	//--------------------------
	//2te Spur am Tag
	//--------------------------
	  //Begin ---------------------------------------------------------------------------------------
	    IF "DB_Schaltuhr".Tag_aktiv[#i].AZ_Begin2_aktiv = true THEN //Wenn Zeit aktiv
	    
	        #Array[#j].Min := TOD_TO_DINT(DTL_TO_TOD("DB_Schaltuhr".Tag[#i].AZ_Begin2))/60000+(#i-1)*1440; //Kopiere im Array
	    #j := #j + 1; //Array+1
	    #pruef := #pruef + 1;
	    
	    IF #anfang = 0 THEN
	        #anfang := 1;
	    END_IF;
	    
	    IF #pruef <> 1 THEN
	        #Error := true;
	    END_IF;
	    
	    END_IF;
	    //Ende ------------------------------------------------------------------------------------------
	    
	    //Begin ---------------------------------------------------------------------------------------
	    IF "DB_Schaltuhr".Tag_aktiv[#i].AZ_Ende2_aktiv = true THEN//Wenn Zeit aktiv
	    
	        #Array[#j].Min := TOD_TO_DINT(DTL_TO_TOD("DB_Schaltuhr".Tag[#i].AZ_Ende2))/60000+(#i-1)* 1440;//Kopiere im Array
	    #j := #j + 1;//Array+1
	    #pruef := #pruef - 1;
	    
	    IF #anfang = 0 THEN
	        #anfang := -1;
	        #pruef := 0; //Pruefparameter wieder auf Null
	    END_IF;
	    
	    IF #pruef <> 0 THEN
	        #Error := true;
	    END_IF;
	    
	    END_IF;
	    //Ende ------------------------------------------------------------------------------------------
	
	 END_FOR;
	 
	//Array schließen ----------------------------
	#Array[#j].Min := -1; //Ende des Arrays
	
	//Plausibilitätsprüfung
	FOR #i:=0 TO #j-2 DO
	  IF #Array[#i+1].Min<=#Array[#i].Min THEN
	    #Error:=true;
	    END_IF;
	  END_FOR;
	
	  IF #anfang = 1 AND #pruef <> 0 OR #anfang = -1 AND #pruef <> 1 OR #anfang=0 THEN //Letzte prüfung
	      #Error := true;
	    END_IF;
	    
	  IF #anfang = -1 THEN //Start mit Ausschaltung
	      #Start_Aus := true;
	  END_IF;
	
	END_IF;
	
END_FUNCTION

FUNCTION_BLOCK "Uhrzeit_WSU"
{ S7_Optimized_Access := 'FALSE' }
VERSION : 0.1
   VAR 
      aktDatum {InstructionName := 'DTL'; LibVersion := '1.0'} : DTL;
      Time_to_on : Int;   // Zeit bis/seit Arbeitszeitbeginn Wert>0-->bis Wert<0-->seit (in Minuten]
      Time_to_off : Int;   // Zeit bis/seit Arbeitszeitende Wert>0-->bis Wert<0-->seit (in Minuten]
      min_of_week : Int;   // Minuten seit Wochenbeginn
      BA_Uhr_Ein : Bool;   // Dauer-Ein BA_Uhr_Aus: 9.0=0 UND 9.1=0
      BA_Uhr_Dauer : Bool;   // Uhrenbetrieb
      AZ_aktiv : Bool;   // Arbeitszeit aktiv
      ProfileWeek : Array[0..28] of Struct   // Wochenschaltpunkte
         MinWeek : Int;
         State : Byte;   // 0=kein Eintrag, bit0=ein, bit1=aus
         resB : Byte;
      END_STRUCT;
   END_VAR

   VAR_TEMP 
      retVal : Int;
      Woko : DInt;   // muss direkt hinter ProfileWeek stehen!
      rdRetval : Int;
      WoTime_bis : Int;
      WoTime_seit : Int;
      TempTime : Int;
      lastOn : Bool;
      nextOn : Bool;
      lastFnd : Bool;
      nextFnd : Bool;
      i : Int;
   END_VAR

   VAR CONSTANT 
      MaxWeek : Int := 10080;   // Anzahl Minuten pro Woche
      "0x7FFF" : Int := 32767;
   END_VAR


BEGIN
	//Lokalzeit auslesen
	IF RD_LOC_T(#aktDatum) > #"0x7FFF"  THEN //Wenn Retval >= 0x08000,
	    RETURN;
	END_IF;
	
	//-------------
	//Betriebsart
	//-------------
	
	//-----------------------------
	//Uhrenbetrieb (Wochenfunktion)
	//-----------------------------
	IF #BA_Uhr_Ein THEN
	    REGION Woche
	        #lastFnd := FALSE;  //letzter Eintrag gefunden/Wochenwechsel erkannt
	        #nextFnd := FALSE;  //nächster Eintrag gefunden
	        #lastOn := FALSE;
	        #nextOn := FALSE;
	        
	        #WoTime_bis := 32767;
	        #WoTime_seit := 32767;
	        
	        //--------------------------------------------------------------------------
	        //Berechnung Minuten seit Wochenbeginn
	        //--------------------------------------------------------------------------
	        #min_of_week := ((USINT_TO_INT(#aktDatum.WEEKDAY) - 1) * 1440) + (USINT_TO_INT(#aktDatum.HOUR) * 60) + USINT_TO_INT(#aktDatum.MINUTE); //Wenn aktueller Wochentag 1 = Sonntag
	        
	        //Schaltuhr leer?
	        IF #ProfileWeek[1].State = b#16#0 THEN
	            #Time_to_on := 32767;
	            #Time_to_off := -32767;
	            
	            //----------------------------
	            //Schaltpunkte suchen
	            //----------------------------
	        ELSE
	            
	            //--------------------------------------------------------------------------
	            //letzten Schaltpunkt suchen
	            //--------------------------------------------------------------------------
	        REGION last
	            //alles ab rela:
	            //vorherigen Schaltpunkt suchen
	                #Woko := #min_of_week;
	                #i := -1;
	                
	                REPEAT //FOR Schleife geht nicht weil ich #i während des Ablaufs nicht verändern darf :-(
	                    
	                    #i += 1;
	                    
	                    IF #ProfileWeek[#i].State <> 0 AND #Woko >= #ProfileWeek[#i].MinWeek THEN //Eintrag leer oder in der Zukunft? dann weiter
	                        //Eintrag gefunden
	                        #lastFnd := TRUE;
	                        IF #ProfileWeek[#i].State = 1 THEN
	                            #lastOn := TRUE;
	                        ELSIF #ProfileWeek[#i].State = 2 THEN
	                            #lastOn := FALSE;
	                        END_IF;
	                        
	                        IF #min_of_week < #ProfileWeek[#i].MinWeek THEN
	                            #WoTime_seit := #MaxWeek - #ProfileWeek[#i].MinWeek + #min_of_week;
	                        ELSE
	                            #WoTime_seit := #min_of_week - #ProfileWeek[#i].MinWeek;
	                        END_IF;
	                    END_IF;
	                    
	                //Prüfung im letzten Durchgang
	                IF #i = 28 THEN
	                    //fündig geworden?
	                    IF #lastFnd THEN//gefunden, ok
	                        EXIT;
	                        
	                    //keinen letzten Schaltpunkt entdeckt
	                    //aktueller Status bleibt erhalten
	                    ELSIF #Woko = #MaxWeek THEN //im 2ten Durchgang?
	                        IF #Time_to_on < 0 THEN
	                            #lastOn := TRUE;
	                            #WoTime_seit := #Time_to_on * -1;
	                        ELSE
	                            #lastOn := FALSE;
	                            #WoTime_seit := #Time_to_off * -1;
	                        END_IF;
	                        
	                        EXIT;
	                        
	                    ELSE//im ersten Durchgang nichts gefunden, dann evtl. in voriger Woche im 2ten Durchgang?
	                        #Woko := #MaxWeek;
	                        #i := -1;
	                    END_IF;
	                END_IF;
	                
	            UNTIL #i = 28
	            END_REPEAT;
	        END_REGION
	            
	            //--------------------------------------------------------------------------
	            //nächsten Schaltpunkt suchen
	            //--------------------------------------------------------------------------
	        REGION next
	            //alles ab snex:
	            //nächsten Schaltpunkt suchen
	            #i := -1;
	            
	            REPEAT //FOR Schleife geht nicht weil ich #i während des Ablaufs nicht verändern darf :-(
	                
	                #i += 1;
	                
	                IF #ProfileWeek[#i].State <> 0 AND #ProfileWeek[#i].MinWeek - #min_of_week >= 0 THEN //Eintrag leer oder in der Zukunft? dann weiter
	                    //Eintrag gefunden
	                    #TempTime := #ProfileWeek[#i].MinWeek - #min_of_week;
	                    
	                    #nextFnd := TRUE;
	                    
	                    IF #TempTime > #WoTime_bis THEN
	                        EXIT;
	                    END_IF;
	                    
	                    #WoTime_bis := #TempTime;
	                    
	                    IF #ProfileWeek[#i].State = 1 THEN
	                        #nextOn := TRUE;
	                    ELSIF #ProfileWeek[#i].State = 2 THEN
	                        #nextOn := FALSE;
	                    END_IF;
	                    EXIT;
	                    
	                END_IF;
	                
	            UNTIL #i = 28
	            END_REPEAT;
	            
	            //nichts gefunden? Dann nächste Woche checken (ersten Eintrag)
	            //Prüfung im letzten Durchgang
	            IF NOT #nextFnd THEN
	                #TempTime := #MaxWeek - #min_of_week + #ProfileWeek[0].MinWeek;
	                #nextFnd := TRUE;
	                IF #TempTime <= #WoTime_bis THEN
	                    #WoTime_bis := #TempTime;
	                    
	                    IF #ProfileWeek[0].State = 1 THEN
	                        #nextOn := TRUE;
	                    ELSIF #ProfileWeek[0].State = 2 THEN
	                        #nextOn := FALSE;
	                    END_IF;
	                END_IF;
	            END_IF;
	            
	        END_REGION
	        
	            END_IF;
	            
	            //Auswertung zum Schluss
	            IF #lastOn AND #nextOn THEN
	                #Time_to_on := 0;// -32767;
	                #Time_to_off := 32767;
	            ELSIF NOT #lastOn AND NOT #nextOn THEN
	                #Time_to_on := 32767;
	                #Time_to_off := 0;// -32767;
	            ELSIF #lastOn AND NOT #nextOn THEN
	                #Time_to_off := #WoTime_bis;
	                #Time_to_on := #WoTime_seit * -1;
	            ELSE
	                #Time_to_on := #WoTime_bis;
	                #Time_to_off := #WoTime_seit * -1;
	            END_IF;
	            
	            
	            
	    END_REGION
	    
	//-----------------------------   
	//Dauerbetrieb
	//-----------------------------
	ELSIF #BA_Uhr_Dauer THEN
	    REGION Dauer
	        #Time_to_on := -32767;
	        #Time_to_off := 32767;
	    END_REGION
	    
	//-----------------------------
	//Aus
	//-----------------------------
	ELSE
	    REGION Aus
	        #Time_to_on := 32767;
	        #Time_to_off := -32767;
	    END_REGION
	END_IF;
	
	//Auswertung Arbeitszeit
	#AZ_aktiv := #Time_to_on <= 0;
	
END_FUNCTION_BLOCK

FUNCTION "Komm_PNOZ" : Void   // FC360, STL
TITLE = Kommunikation Pilz-PNOZ <--> PLC
{ S7_Optimized_Access := 'FALSE' }
// stored: AutoNumber false
   VAR_TEMP
      Checksum : Word;
      ReturnValue : Int;
      count : Byte;
   END_VAR
BEGIN

NETWORK
TITLE = Aktivierung der Kommunikation

      AN    "DB_PNOZ_Comm".connection.activate;
      A     "E_T_ErrQ";
      S     "DB_PNOZ_Comm".connection.activate;


NETWORK
TITLE = OUTPUT --> PNOZ
// siehe Handbuch
// "PNOZmulti_2_Com_Interf_Man_1002971-de-03.pdf"
// Set Header   (Kap. 5.5)
      L     16#05;
      T     "DB_PNOZ_IN_Out".Out.Header[0];

      L     16#15;
      T     "DB_PNOZ_IN_Out".Out.Header[1];

      L     16#00;
      T     "DB_PNOZ_IN_Out".Out.Header[2];

      L     16#26;  // Anzahl Nutzdaten +5  = 38 dez
      T     "DB_PNOZ_IN_Out".Out.Header[3];

      L     16#5C;  // Anforderungs-Nr
      T     "DB_PNOZ_IN_Out".Out.Header[4];

      L     16#00;
      T     "DB_PNOZ_IN_Out".Out.Header[5];  // Control Byte Bit 0..2 Watchdog

      L     16#00;
      T     "DB_PNOZ_IN_Out".Out.Header[6];

      L     16#00;  // immer 0x00
      T     "DB_PNOZ_IN_Out".Out.Header[7];

      L     16#10;
      T     "DB_PNOZ_IN_Out".Out.Endekennung;

// Set Vitual OUTput - je nach Projekt
      A     "E_T_Q_Not-Halt";
// alle Schütze müssen abgefallen sein
      A     "E_RM_NH_Dkl";
      A     "E_RM_NH_FP_CM01.GP01";
      A     "E_RM_NH_FP_CM01.GP04";
      A     "E_RM_NH_Pumpen";
      =     "DB_PNOZ_IN_Out".Out.T_NH_Quitt;
// Freigabe Automatik
      A     "E_Frg_Auto";
      =     "DB_PNOZ_IN_Out".Out.Frg_Automatik;

      CLR;
      =     "DB_PNOZ_IN_Out".Out.VirtualOutput[16];
// ...
      =     "DB_PNOZ_IN_Out".Out.VirtualOutput[127];

// Berechnung der Checksumme (4+ .. 39)

      LAR1  P#48.0;  // fix 44 (IN) + 4

      L     "DB_PNOZ_IN_Out".Out.Header[4];  //Start
      T     #Checksum;

      L     35;  // fix: 39 - 4
T_CS: T     #count;
      OPN   "DB_PNOZ_IN_Out";
      +AR1  P#1.0;
      L     #Checksum;
      L     DBB [AR1, P#0.0];
      +I;
      T     #Checksum;

      L     #count;  //Schleifenzähler
      LOOP  T_CS;

      L     16#00;
      L     #Checksum;
      AW    16#00FF;
      -I;
      T     "DB_PNOZ_IN_Out".Out.Checksum;



NETWORK
TITLE = Umkopieren
// Sende-/Empfangsdaten umkopieren

      A     "DB_PNOZ_Comm".RECEIVE.NDR;
      R     "DB_PNOZ_Comm".RECEIVE.NDR;
      JCN   Send;

      CALL  BLKMOV
      ( SRCBLK  := "DB_PNOZ_Receive".In,
        RET_VAL := #ReturnValue,
        DSTBLK  := "DB_PNOZ_IN_Out".In
      );

Send: A     "DB_PNOZ_Comm".SEND.Busy;
      JC    no_Send_DATA;

      CALL  BLKMOV
      ( SRCBLK  := "DB_PNOZ_IN_Out".Out,
        RET_VAL := #ReturnValue,
        DSTBLK  := "DB_PNOZ_Send".Out
      );

no_Send_DATA:NOP   0;

NETWORK
TITLE = Sprungverteiler

      L     "DB_PNOZ_Comm".Global_Status;
      JL    LSTX;
      JU    OFF;  // 0: Aus
      JU    CONN;  // 1: Verbindungsaufbau
      JU    WRIT;  // 2: Schreiben
      JU    READ;  // 3: Lesen
      JU    DISC;  // 4:Verbindungsabbau
      JU    ERR;  // 5: Fehler
LSTX: JU    ende;

//*
// wait for user input (activate / deactivate communication)
// - if activate change for 0 to 1
//    => status is set to 1 (connect) and all status-values are set to default
// - if activate change for 1 to 0
//    => status is set to 4 (disconnect)
//-

OFF:  A     "DB_PNOZ_Comm".connection.activate;
      AN    "DB_PNOZ_Comm".connection.established;
      JCN   OFF1;

// Aktivieren
      SET;
      S     "DB_PNOZ_Comm".connection.established;

      L     1;  // Verbindungsaufbau
      T     "DB_PNOZ_Comm".Global_Status;

// init
      SET;
      R     "DB_PNOZ_Comm".CONNECT.Request;
      R     "DB_PNOZ_Comm".CONNECT.Done;
      R     "DB_PNOZ_Comm".CONNECT.Error;

      R     "DB_PNOZ_Comm".SEND.Request;
      R     "DB_PNOZ_Comm".SEND.Done;
      R     "DB_PNOZ_Comm".SEND.Error;

      S     "DB_PNOZ_Comm".RECEIVE.EN_R;  // immer 1
      R     "DB_PNOZ_Comm".RECEIVE.NDR;
      R     "DB_PNOZ_Comm".RECEIVE.Error;

      R     "DB_PNOZ_Comm".DISCONNECT.Request;
      R     "DB_PNOZ_Comm".DISCONNECT.Done;
      R     "DB_PNOZ_Comm".DISCONNECT.Error;

      JU    ende;

// Deaktivieren
OFF1: AN    "DB_PNOZ_Comm".connection.activate;
      A     "DB_PNOZ_Comm".connection.established;
      JCN   ende;

      SET;
      R     "DB_PNOZ_Comm".connection.established;
      R     "DB_PNOZ_Comm".CONNECT.Done;
      R     "DB_PNOZ_Comm".SEND.Done;
      R     "DB_PNOZ_Comm".RECEIVE.NDR;

      L     4;  // Verbindungsabbau
      T     "DB_PNOZ_Comm".Global_Status;

      JU    ende;


NETWORK
TITLE = Verbindungsaufbau
// call FB65 (TCON) as long as status = 1 (connect)
//  - if connection_1 is established (TCON_DONE=1) change to status=2 (send)
//  - if an error occurs (TCON_ERR=1) change to status=5 (error)
CONN: L     2;
      T     "DB_PNOZ_Comm".CONNECT.ID;
      T     "DB_PNOZ_Comm".Connection_Param.local_device_id;

      CALL  TCON, "TCON_DI"
      ( REQ     := "DB_PNOZ_Comm".CONNECT.Request,
        ID      := "DB_PNOZ_Comm".CONNECT.ID,
        DONE    := "DB_PNOZ_Comm".CONNECT.Done,
        BUSY    := "DB_PNOZ_Comm".CONNECT.Busy,
        ERROR   := "DB_PNOZ_Comm".CONNECT.Error,
        STATUS  := "DB_PNOZ_Comm".CONNECT.Status,
        CONNECT := "PNOZ_Connection_DB"
      );

      SET;
      S     "DB_PNOZ_Comm".CONNECT.Request;

      A     "DB_PNOZ_Comm".CONNECT.Done;
      R     "DB_PNOZ_Comm".CONNECT.Done;
      R     "DB_PNOZ_Comm".SEND.Request;
      JC    to_S;

      L     "DB_PNOZ_Comm".CONNECT.Status;
      L     16#80A3;  //Verbindung gibt's schon
      ==I;
      A     "DB_PNOZ_Comm".CONNECT.Error;
      R     "DB_PNOZ_Comm".DISCONNECT.Request;
      JC    to_D;

      A     "DB_PNOZ_Comm".CONNECT.Error;
      JC    to_E;

      JU    ende;

to_S: L     2;  // --> Senden
      T     "DB_PNOZ_Comm".Global_Status;
      JU    ende;

to_D: L     4;  // --> Verbindungsabbau
      T     "DB_PNOZ_Comm".Global_Status;
      JU    ende;


to_E: L     5;  // --> Fehler
      T     "DB_PNOZ_Comm".Global_Status;

      JU    ende;


NETWORK
TITLE = Schreiben --> PNOZ
// call FB63 (TSEND) as long as status = 2 (send)
//  - if send is complete (TSEND_DONE=1) change to status=3 (receive)
//  - if an error occurs (TSEND_ERR=1)
//    - if TSEND_STATUS='80A1' or '80C4' stay at status=2 and try to send again
//    - if TSEND_STATUS<>'80A1' or '80C4' change to status=5 (error)
WRIT: L     43;  //fix PNOZ
      T     "DB_PNOZ_Comm".SEND.Length;

      L     "DB_PNOZ_Comm".CONNECT.ID;
      T     "DB_PNOZ_Comm".SEND.ID;

      CALL  TSEND, "TSEND_DI"
      ( REQ    := "DB_PNOZ_Comm".SEND.Request,
        ID     := "DB_PNOZ_Comm".SEND.ID,
        LEN    := "DB_PNOZ_Comm".SEND.Length,
        DONE   := "DB_PNOZ_Comm".SEND.Done,
        BUSY   := "DB_PNOZ_Comm".SEND.Busy,
        ERROR  := "DB_PNOZ_Comm".SEND.Error,
        STATUS := "DB_PNOZ_Comm".SEND.Status,
        DATA   := "DB_PNOZ_Send".Out
      );

      SET;
      S     "DB_PNOZ_Comm".SEND.Request;

      A     "DB_PNOZ_Comm".SEND.Done;
      R     "DB_PNOZ_Comm".SEND.Done;
      S     "DB_PNOZ_Comm".RECEIVE.EN_R;
      JC    toRV;

      L     16#80A1;  //Kommunikationsfehler
      L     "DB_PNOZ_Comm".SEND.Status;
      ==I;
      O(;
      L     16#80C4;  //Temporärer Kommunikationsfehler
      ==I;
      );
      A     "DB_PNOZ_Comm".SEND.Error;
      R     "DB_PNOZ_Comm".SEND.Request;  // --> nochmal versuchen
      JC    ende;

      A     "DB_PNOZ_Comm".SEND.Error;
      JC    SDER;

      JU    ende;

toRV: L     3;
      T     "DB_PNOZ_Comm".Global_Status;
      JU    ende;

SDER: L     5;
      T     "DB_PNOZ_Comm".Global_Status;
      JU    ende;


NETWORK
TITLE = Lesen <-- PNOZ
// call FB64 (TRCV) as long as status = 3 (receive)
//  - if new data is received (TSEND_NDR=1) change to status=2 (receive)
//    and increment send_values
//  - if an error occurs (TRCV_ERR=1)
//    - if TRCV_STATUS='80A1' or '80C4' change to status=2 and try to send
//    - if TRCV_STATUS<>'80A1' or '80C4' change to status=5 (error)
READ: L     43;  //fix PNOZ
      T     "DB_PNOZ_Comm".RECEIVE.Length;

      L     "DB_PNOZ_Comm".CONNECT.ID;
      T     "DB_PNOZ_Comm".RECEIVE.ID;

      CALL  TRCV, "TRCV_DI"
      ( EN_R     := "DB_PNOZ_Comm".RECEIVE.EN_R,
        ID       := "DB_PNOZ_Comm".RECEIVE.ID,
        LEN      := "DB_PNOZ_Comm".RECEIVE.Length,
        ADHOC    := "DB_PNOZ_Comm".RECEIVE.ADHOC,
        NDR      := "DB_PNOZ_Comm".RECEIVE.NDR,
        BUSY     := "DB_PNOZ_Comm".RECEIVE.Busy,
        ERROR    := "DB_PNOZ_Comm".RECEIVE.Error,
        STATUS   := "DB_PNOZ_Comm".RECEIVE.Status,
        RCVD_LEN := "DB_PNOZ_Comm".RECEIVE.Receive_Length,
        DATA     := "DB_PNOZ_Receive".In
      );

      A     "DB_PNOZ_Comm".RECEIVE.NDR;
      JC    toSD;

      L     16#80A1;  //Kommunikationsfehler
      L     "DB_PNOZ_Comm".RECEIVE.Status;
      ==I;
      O(;
      L     16#80C4;  //Temporärer Kommunikationsfehler
      ==I;
      );
      A     "DB_PNOZ_Comm".RECEIVE.Error;
      R     "DB_PNOZ_Comm".RECEIVE.Error;
      JC    toSD;

      A     "DB_PNOZ_Comm".RECEIVE.Error;
      JC    RVER;

      JU    ende;

toSD: L     2;
      T     "DB_PNOZ_Comm".Global_Status;
      SET;
      R     "DB_PNOZ_Comm".SEND.Request;
      JU    ende;

RVER: L     5;
      T     "DB_PNOZ_Comm".Global_Status;
      JU    ende;


NETWORK
TITLE = Verbindungsabbau
// call FB66 (TDISCON) as long as status = 4 (disconnect)
//  - if connection_1 is disconnected (TDISCON_DONE=1) change to status=0 (init)
//  - if an error occurs (TDISCON_ERR=1) change to status=5 (error)
DISC: L     "DB_PNOZ_Comm".CONNECT.ID;
      T     "DB_PNOZ_Comm".DISCONNECT.ID;

      CALL  TDISCON, "TDISCON_DI"
      ( REQ    := "DB_PNOZ_Comm".DISCONNECT.Request,
        ID     := "DB_PNOZ_Comm".DISCONNECT.ID,
        DONE   := "DB_PNOZ_Comm".DISCONNECT.Done,
        BUSY   := "DB_PNOZ_Comm".DISCONNECT.Busy,
        ERROR  := "DB_PNOZ_Comm".DISCONNECT.Error,
        STATUS := "DB_PNOZ_Comm".DISCONNECT.Status
      );

      SET;
      S     "DB_PNOZ_Comm".DISCONNECT.Request;

      A     "DB_PNOZ_Comm".DISCONNECT.Done;
      R     "DB_PNOZ_Comm".DISCONNECT.Done;
      R     "DB_PNOZ_Comm".connection.activate;
      R     "DB_PNOZ_Comm".connection.established;
      JC    to_O;

      A     "DB_PNOZ_Comm".DISCONNECT.Error;
      JC    toE;

      JU    ende;

to_O: L     0;  // --> OFF
      T     "DB_PNOZ_Comm".Global_Status;
      JU    ende;

toE:  L     5;  // --> Fehler
      T     "DB_PNOZ_Comm".Global_Status;
      JU    ende;


NETWORK
TITLE = Fehler
ERR:  SET;
      R     "DB_PNOZ_Comm".connection.activate;
      R     "DB_PNOZ_Comm".connection.established;

      L     0;  // --> OFF
      T     "DB_PNOZ_Comm".Global_Status;

ende: BE;

END_FUNCTION

FUNCTION "FC_DP_Error" : Void   // FC203, STL
TITLE = Profibusfehler melden
{ S7_Optimized_Access := 'FALSE' }
// stored: AutoNumber false
   VAR_TEMP
      RetVal : Int;
      Adresse : DWord;
      Count : Int;
      Wert_akt : Byte;
      Wert_alt : Byte;
      Err_Nr : USInt;
      Inf : Struct
         Inf1 : Byte;
         inf2 : Byte;
      END_STRUCT;
   END_VAR
BEGIN

NETWORK
TITLE = Störung/Ausfall
      AN    "DB_ANLAGE".config.Check_Profibus;  //keine Überwachung gefordert
      ON    "DB_ANLAGE".IN.Watch_Profibus;  //Überwachung nicht möglich
      BEC;
      R     "DB_DP_Error".Sammelwarnung;
      R     "DB_DP_Error".Sammelstoerung;

      A     "DB_ANLAGE".IN.PC_offline;  //kein PC-aktiv --> keine Überwachung
      BEC;

//Erstmalige Prüfung?
      AN    "DB_DP_Error".Init;
      AN    "DB_ANLAGE".IN.AMS_Restart;
      JC    norm;


NETWORK
TITLE = erstmalige Prüfung --> nur Fehlerstatus 2oder 3 senden
// Statuswert Bedeutung:
// 0: nicht projektiert & nicht vorhanden
// 1: vorhanden & ok
// 2: vorhanden aber nicht ok
// 3: projektiert aber nicht vorhanden
      SET;
      R     "DB_DP_Error".Init;

//aktuellen Status als Altstatus übernehmen
      CALL  FILL
      ( BVAL    := "DB_DP_Error".DP_Slave,
        RET_VAL := #RetVal,
        BLK     := "DB_DP_Error".Altwert
      );

//Altwert-Einträge mit Status 0,1 bleiben
//Einträge mit 2,3 werden auf 1 gesetzt
//dadurch wird bei fehlerhaften Einträgen ein Wechsel von 1 auf 2 oder 3 erkannt
//und somit erneut gemeldet
      L     0;
      L     "DB_DP_Error".HiAdr;
      ==I;
      BEC;
retC: T     #Count;
      L     1024;
      +D;
      SLD   3;
      T     #Adresse;
      OPN   "DB_DP_Error";
      L     DBB [#Adresse];
      L     1;  //Wert 0,1 bleibt erhalten
      <=I;
      JC    nexC;
      T     DBB [#Adresse];
nexC: L     #Count;
      LOOP  retC;  //Wert 2,3 mit 1 überschreiben

NETWORK
TITLE = Normalprüfung --> jede Statusänderung melden
norm: NOP   0;

      L     0;  //keine Profibusteilnehmer
      L     "DB_DP_Error".HiAdr;
      ==I;
      BEC;
reC:  T     #Count;
      SLD   3;
      T     #Adresse;
      OPN   "DB_DP_Error";
      L     DBB [#Adresse];
      T     #Wert_akt;  //"DB_DP_Error".DP_Slave[#Count]

      L     #Wert_akt;  //Warnung melden
      L     2;
      ==I;
      S     "DB_DP_Error".Sammelwarnung;
      L     #Wert_akt;  //Störung melden
      L     3;
      ==I;
      S     "DB_DP_Error".Sammelstoerung;

      L     #Count;
      +     1024;
      SLD   3;
      T     #Adresse;
      OPN   "DB_DP_Error";
      L     DBB [#Adresse];
      T     #Wert_alt;

//Statusauswertung und Änderung melden
      L     #Wert_akt;  //"DB_DP_Error".Altwert[#Count]
      L     #Wert_alt;
      ==I;
      JC    nxC;
      L     #Wert_alt;
      JL    list;
      JU    old0;
      JU    old1;
      JU    old2;
      JU    old3;
list: JU    nxC;

//Baugruppe war weder projektiert noch vorhanden
old0: L     #Wert_akt;
      T     #Err_Nr;
      JC    evt;

//Baugruppe war projektiert und vorhanden
old1: L     0;  //Wechsel auf 0 ist ok
      L     #Wert_akt;
      ==I;
      JC    nxC;
      T     #Err_Nr;
      JC    evt;

//Baugruppe war projektiert,vorhanden aber fehlerhaft
old2: L     0;  //Wechsel auf 0 ist ok
      L     #Wert_akt;
      ==I;
      JC    nxC;
      T     #Err_Nr;
      JC    evt;

//Baugruppe war projektiert aber nicht vorhanden
old3: L     0;  //Wechsel auf 0 ist ok
      L     #Wert_akt;
      ==I;
      JC    nxC;
      T     #Err_Nr;
      JC    evt;

evt:  NOP   0;
//Err_Nr 1:Station wiederkehr
//Err_Nr 2:Station nicht ok
//Err_Nr 3:Station Ausfall
      CALL  BLKMOV
      ( SRCBLK  := #Count,
        RET_VAL := #RetVal,
        DSTBLK  := #Inf
      );


      L     #Err_Nr;
      L     3;
      ==I;
      A     "DB_DP_Error".Hupe_enable;
      R     "DB_ANLAGE".config.M_Q_Hupe;

nxC:  L     #Count;
      LOOP  reC;

//aktuellen Status als Altstatus übernehmen
      CALL  FILL
      ( BVAL    := "DB_DP_Error".DP_Slave,
        RET_VAL := #RetVal,
        BLK     := "DB_DP_Error".Altwert
      );

END_FUNCTION

FUNCTION "FU_Read" : Void
{ S7_Optimized_Access := 'TRUE' }
VERSION : 0.1
   VAR_TEMP 
      i : Int;
      Ret_Value : Int;
   END_VAR


BEGIN
	IF "DB_ANLAGE".BA.Simulation THEN
	    RETURN;
	END_IF;
	
	// Pumpen
	#Ret_Value := DPRD_DAT(LADDR := "SEW-GW_UC01~Filterbeschickung_HQ01", RECORD => "FU_In_Out".FU[1].PE);
	#Ret_Value := DPRD_DAT(LADDR := "SEW-GW_UC01~Umwaelzung_CM01", RECORD => "FU_In_Out".FU[2].PE);
	#Ret_Value := DPRD_DAT(LADDR := "SEW-GW_UC01~Umwaelzung_CM03", RECORD => "FU_In_Out".FU[3].PE);
	#Ret_Value := DPRD_DAT(LADDR := "SEW-GW_UC01~Filterbeschickung_HQ02", RECORD => "FU_In_Out".FU[4].PE);
	#Ret_Value := DPRD_DAT(LADDR := "SEW-GW_UC01~Umwaelzung_CM02", RECORD => "FU_In_Out".FU[5].PE);
	#Ret_Value := DPRD_DAT(LADDR := "SEW-GW_UC01~Umwaelzung_CM04", RECORD => "FU_In_Out".FU[6].PE);
	//Ventilator
	#Ret_Value := DPRD_DAT(LADDR := "SEW-GW_UC01~Ventilator_Sperrluft", RECORD => "FU_In_Out".FU[7].PE);
	
	// QF
	#Ret_Value := DPRD_DAT(LADDR := "SEW-GW_UC06~QF_WR02", RECORD => "FU_In_Out".FU[8].PE);
	#Ret_Value := DPRD_DAT(LADDR := "SEW-GW_UC06~QF_WR03", RECORD => "FU_In_Out".FU[9].PE);
	// TW
	#Ret_Value := DPRD_DAT(LADDR := "SEW-GW_UC07~TW_Fahrt", RECORD => "FU_In_Out".FU[10].PE);
	#Ret_Value := DPRD_DAT(LADDR := "SEW-GW_UC07~TW_Hub_li_WR04", RECORD => "FU_In_Out".FU[11].PE);
	#Ret_Value := DPRD_DAT(LADDR := "SEW-GW_UC07~TW_Hub_re_WR05", RECORD => "FU_In_Out".FU[12].PE);
	
	FOR #i := 1 TO "FU_In_Out".Anzahl DO
	    IF "DB_ANLAGE".IN.Quitt_Err THEN
	        "FU_In_Out".FU[#i].Fehler := FALSE;
	    END_IF;
	    
	    "FU_In_Out".FU[#i].Fehler := "FU_In_Out".FU[#i].PE.Statusbyte.Stoer;
	    "FU_In_Out".FU[#i].AM_Fehlernummer := "FU_In_Out".FU[#i].PE.Statusbyte.Fehlernummer;
	END_FOR;
	
	
END_FUNCTION

FUNCTION "FC_INPUT" : Void   // FC210, STL
TITLE = Einlesen der physikalischen Eingänge
{ S7_Optimized_Access := 'FALSE' }
AUTHOR : RE
// stored: AutoNumber false
   VAR_TEMP
      WT_DB : Int;
      RetVal : Int;
   END_VAR
   VAR CONSTANT
      Aufgabe_KS : USInt := 1;
      Aufgabe_LS : USInt := 2;
      Aufgabe_GO : USInt := 3;
   END_VAR
BEGIN

NETWORK
TITLE = Simulation
// Adressen für Diagnose sind in der Hardware-Konfiguration
// hinterlegt und sind noch anzupassen !!!

//---------------------------------------------------
//Fehlerquittung
      A     "E_T_ErrQ";
      O     "MobilePanel".Drucktaster_K2_Push;
      FP    "DB_ANLAGE".config.FP_In_Quitt;
      =     "DB_ANLAGE".IN.Quitt_Err;
      L     s5t#500ms;
      Extend "T_ErrQuitt";

//---------------------------------------------------


NETWORK
TITLE = Einlesen Digitale Eingäne (allgemein)
ok:   SET;

      AN    "DB_PNOZ_IN_Out".In.PNOZ_OK;
      =     "DB_ANLAGE".IN.S_Not_Aus;

NoQt: SET;
      =     "DB_ANLAGE".IN.S_St_Spng;
      A     "E_T_HupeQ";
      =     "DB_ANLAGE".IN.Quitt_Hupe;
      =     "DB_Alarme".IN_Quitt_Hupe;

//Reperaturbetrieb über Schlüssel-Panel
      A     "MobilePanel".Koordinierung.%X2;
      L     S5T#2s;
      SD    "T_MobielPanel_Lebensbit_ein";

      AN    "MobilePanel".Koordinierung.%X2;
      L     S5T#2s;
      SD    "T_MobielPanel_Lebensbit_aus";

      A     "MobilePanel".Schluessel;
      S     "DB_ANLAGE".IN.Reparatur;

      AN    "MobilePanel".Schluessel;
      O     "T_MobielPanel_Lebensbit_ein";
      O     "T_MobielPanel_Lebensbit_aus";
      R     "DB_ANLAGE".IN.Reparatur;

      CLR;
      =     "DB_ANLAGE".IN.Reset;
      =     "DB_ANLAGE".IN.Lamp_Test;

      A     "E_Frg_Auto";
      O     "DB_ANLAGE".BA.Simulation;
      R     "DB_ANLAGE".IN.BA_Tipp;
      R     "DB_ANLAGE".IN.BA_Hand;
      S     "DB_ANLAGE".IN.BA_Auto;

      AN    "E_Frg_Auto";
      A     "Panel".Betriebsart.Hand;
      R     "DB_ANLAGE".IN.BA_Tipp;
      S     "DB_ANLAGE".IN.BA_Hand;
      R     "DB_ANLAGE".IN.BA_Auto;

      AN    "E_Frg_Auto";
      A     "Panel".Betriebsart.Tipp;
      S     "DB_ANLAGE".IN.BA_Tipp;
      R     "DB_ANLAGE".IN.BA_Hand;
      R     "DB_ANLAGE".IN.BA_Auto;

      A     "DB_ANLAGE".IN.BA_Auto;
      A     "Panel".Betriebsart.Automatik;
      R     "DB_ANLAGE".IN.Automat_aus;
      S     "DB_ANLAGE".IN.Automat_ein;

      AN    "E_Frg_Auto";
      ON    "Panel".Betriebsart.Automatik;
      S     "DB_ANLAGE".IN.Automat_aus;
      R     "DB_ANLAGE".IN.Automat_ein;

      L     1;
      A     "DB_ANLAGE".config.NormalB;
      =     "Panel".Betriebsmodus.Normal;
      R     "Panel".Betriebsmodus.Kombi;
      JC    A_BM;
      L     2;
      AN    "DB_ANLAGE".config.NormalB;
      =     "Panel".Betriebsmodus.Kombi;
      R     "Panel".Betriebsmodus.Normal;

A_BM: T     "Panel".Betriebsmodus.Anzeige;
// Wechsel nur bei komplett leerer Anlage
      L     "DI_FW_1".ZST.WT_DB_NR_li;
      L     0;
      ==I;
      A(;
      L     "DI_FW_1".ZST.WT_DB_NR_re;
      ==I;
      );
      AN    "DB_POS".POS[1].belegt;
      AN    "DB_POS".POS[2].belegt;
      AN    "DB_POS".POS[3].belegt;
      AN    "DB_POS".POS[4].belegt;
      AN    "DB_POS".POS[5].belegt;
      AN    "DB_POS".POS[6].belegt;
      AN    "DB_POS".POS[7].belegt;
      AN    "DB_POS".POS[8].belegt;
      AN    "DB_POS".POS[9].belegt;
      AN    "DB_POS".POS[10].belegt;
      AN    "DB_POS".POS[11].belegt;
      AN    "DB_POS".POS[12].belegt;
      AN    "DB_POS".POS[13].belegt;
      AN    "DB_POS".POS[14].belegt;
      AN    "DB_POS".POS[15].belegt;
      AN    "DB_POS".POS[16].belegt;
      AN    "DB_POS".POS[17].belegt;
      AN    "DB_POS".POS[18].belegt;
      AN    "DB_POS".POS[19].belegt;
      AN    "DB_POS".POS[20].belegt;
      AN    "DB_POS".POS[21].belegt;
      AN    "DB_POS".POS[22].belegt;
      AN    "DB_POS".POS[23].belegt;
      AN    "DB_POS".POS[24].belegt;
      AN    "DB_POS".POS[25].belegt;
      AN    "DB_POS".POS[26].belegt;
      AN    "DB_POS".POS[27].belegt;
      AN    "DB_POS".POS[28].belegt;
      AN    "DB_POS".POS[29].belegt;
      AN    "DB_POS".POS[30].belegt;
      AN    "DB_BE_Stand".Stand[1].IN_Belegt;
      AN    "DB_BE_Stand".Stand[2].IN_Belegt;
      AN    "DB_BE_Stand".Stand[3].IN_Belegt;
      AN    "DB_BE_Stand".Stand[4].IN_Belegt;
      AN    "DB_BE_Stand".Stand[5].IN_Belegt;
      AN    "DB_BE_Stand".Stand[6].IN_Belegt;
      =     "Panel".Betriebsmodus.Wechsel_erlaubt;


NETWORK
TITLE = Transportsystem Fahrwagen
      L     S5T#2S;
      A     "DB_ANLAGE".IN.S_Not_Aus;
      SF    "T_Verz_NotAus";
//--------------------------
//Fernbedienung
//--------------------------
// --> Mobile Panel

//--------------------------
//Kollision FW
//--------------------------
// nur ein TW - wird intern gebildet (Wägezellen)

//--------------------------
//Fahrwagen 1
//--------------------------
      A     "T_Verz_NotAus";
      ON    "DB_PNOZ_IN_Out".In.NH_Frg_TW_QF;
      =     "DI_FW_1".ErrIn.Alarm.NotHalt;
      A     "DB_ANLAGE".BA.Tippbetrieb;
      =     "DI_FW_1".IN.BA_Tipp_ext;
      A     "DB_ANLAGE".BA.Handbetrieb;
      =     "DI_FW_1".IN.BA_Hand_ext;
      A     "DB_ANLAGE".BA.Automat_ein;
      =     "DI_FW_1".IN.BA_Auto_ext;
      A     "DB_ANLAGE".BA.Automat_aus;
      =     "DI_FW_1".IN.BA_Auto_Stop_ext;
      A     "DB_ANLAGE".IN.Reparatur;
      =     "DI_FW_1".IN.REP_TASTE;
      A     "DB_ANLAGE".IN.Quitt_Err;
      =     "DI_FW_1".IN.QUITT_ALARM;

      A     "DB_ANLAGE".IN.BA_Tipp;
      S     "DI_FW_1".IN.BA_Tipp_ext;
      R     "DI_FW_1".IN.BA_Hand_ext;
      R     "DI_FW_1".IN.BA_Auto_ext;

// Panel-Tasten

      A     "Panel".TW.T_rueck;
      =     "DI_FW_1".IN.DIR_RCK;
      A     "T_MobielPanel_Lebensbit_ein";
      O     "T_MobielPanel_Lebensbit_aus";
      R     "Panel".TW.T_rueck;

      A     "Panel".TW.T_vor;
      =     "DI_FW_1".IN.DIR_VOR;
      A     "T_MobielPanel_Lebensbit_ein";
      O     "T_MobielPanel_Lebensbit_aus";
      R     "Panel".TW.T_vor;

      A     "Panel".TW.T_heben_li;
      O     "Panel".TW.T_heben;
      =     "DI_FW_1".IN.DIR_HEB_li;
      A     "T_MobielPanel_Lebensbit_ein";
      O     "T_MobielPanel_Lebensbit_aus";
      R     "Panel".TW.T_heben;
      R     "Panel".TW.T_heben_li;

      A     "Panel".TW.T_senken_li;
      O     "Panel".TW.T_senken;
      =     "DI_FW_1".IN.DIR_SENK_li;
      A     "T_MobielPanel_Lebensbit_ein";
      O     "T_MobielPanel_Lebensbit_aus";
      R     "Panel".TW.T_senken;
      R     "Panel".TW.T_senken_li;

      A     "Panel".TW.T_heben_re;
      O     "Panel".TW.T_heben;
      =     "DI_FW_1".IN.DIR_HEB_re;
      A     "T_MobielPanel_Lebensbit_ein";
      O     "T_MobielPanel_Lebensbit_aus";
      R     "Panel".TW.T_heben;
      R     "Panel".TW.T_heben_re;

      A     "Panel".TW.T_senken_re;
      O     "Panel".TW.T_senken;
      =     "DI_FW_1".IN.DIR_SENK_re;
      A     "T_MobielPanel_Lebensbit_ein";
      O     "T_MobielPanel_Lebensbit_aus";
      R     "Panel".TW.T_senken;
      R     "Panel".TW.T_senken_re;

      A     "Panel".TW.T_Halt;
      =     "DI_FW_1".IN.Halt;

      A     "DB_PNOZ_IN_Out".In.T_Aktion_MP;
      O(;
      A     "DB_PNOZ_IN_Out".In.Tuer_VS_ok;
      A     "DB_PNOZ_IN_Out".In.Tuer_RS_ok;
      );
      O     "DB_ANLAGE".BA.Simulation;
      =     "DI_FW_1".IN.Aktion;

      SET;
      S     "DI_FW_1".IN.Knauf_Auto;

      A     "DB_ANLAGE".BA.Simulation;
      BEC;
//===========================================================================
      SET;
      S     "DI_FW_1".ZST.REFERENZIERT;
      R     "DI_FW_1".IN.FahrBreak_on;
      R     "DI_FW_1".IN.HubBreak_on;

// FU[10] - Fahrt
      A     "FU_In_Out".FU[10].PE.Statusbyte.Stoer;
      O(;
      A     "FU_In_Out".FU[10].PA.Steuerwort.FrgStop;
      AN    "FU_In_Out".FU[10].PE.Statusbyte.Bereit;
      );
      AN    "DI_FW_1".ErrIn.Alarm.NotHalt;
      =     "DI_FW_1".ErrIn.Alarm.Fahrt_nok;
// FU[11] - Hub links
      A     "FU_In_Out".FU[11].PE.Statusbyte.Stoer;
      O(;
      A     "FU_In_Out".FU[11].PA.Steuerwort.FrgStop;
      AN    "FU_In_Out".FU[11].PE.Statusbyte.Bereit;
      );
      AN    "DI_FW_1".ErrIn.Alarm.NotHalt;
      =     "DI_FW_1".ErrIn.Alarm.Hub_nok_links;
// FU[12] - Hub rechts
      A     "FU_In_Out".FU[12].PE.Statusbyte.Stoer;
      O(;
      A     "FU_In_Out".FU[12].PA.Steuerwort.FrgStop;
      AN    "FU_In_Out".FU[12].PE.Statusbyte.Bereit;
      );
      AN    "DI_FW_1".ErrIn.Alarm.NotHalt;
      =     "DI_FW_1".ErrIn.Alarm.Hub_nok_rechts;

      CLR;
      =     "DI_FW_1".ErrIn.Warnung.Wrn_Temp_Fahr;
      =     "DI_FW_1".ErrIn.Warnung.Wrn_Temp_Hub;
      =     "DI_FW_1".ErrIn.Alarm.AFS_BS;
      =     "DI_FW_1".ErrIn.Alarm.AFS_WS;
      =     "DI_FW_1".ErrIn.Alarm.POS_BELEGT_li;
      =     "DI_FW_1".ErrIn.Alarm.F_Brk_Fahr;
      =     "DI_FW_1".ErrIn.Alarm.F_Brk_Hub_links;
      =     "DI_FW_1".ErrIn.Alarm.F_Brk_Hub_rechts;

      A     "E_BE_vor_TW";
      =     "DI_FW_1".ErrIn.Alarm.BE_Vor;
      A     "E_BE_rck_TW";
      =     "DI_FW_1".ErrIn.Alarm.BE_Rck;

      A     "E_GurtUeL_li";
      =     "DI_FW_1".ErrIn.Alarm.Gurt_UeL_links;

      A     "E_GurtUeL_re";
      =     "DI_FW_1".ErrIn.Alarm.Gurt_UeL_rechts;

      A     "E_not_unten_li";
      =     "DI_FW_1".ErrIn.Alarm.Gurt_DN_links;
      A     "E_Not_oben_li";
      =     "DI_FW_1".ErrIn.Alarm.Gurt_UP_links;

      A     "E_not_unten_re";
      =     "DI_FW_1".ErrIn.Alarm.Gurt_DN_rechts;
      A     "E_Not_oben_re";
      =     "DI_FW_1".ErrIn.Alarm.Gurt_UP_rechts;

// Lastüberwachung
      A     "A_Heb_li";
      AN    "E_Frg_Heb_li";
      O;
      A     "A_Snk_li";
      AN    "E_Frg_Snk_li";
      L     s5t#200ms;
      SD    "T_St_Last_links";

      A     "T_St_Last_links";
      ON    "E_UeL_ok_li";
      AN    "DI_FW_1".ErrIn.Alarm.NotHalt;
      S     "DI_FW_1".ErrIn.Alarm.Last_UeW_links;

      A     "A_Heb_re";
      AN    "E_Frg_Heb_re";
      O;
      A     "A_Snk_re";
      AN    "E_Frg_Snk_re";
      L     s5t#200ms;
      SD    "T_St_Last_rechts";

      A     "T_St_Last_rechts";
      ON    "E_UeL_ok_re";
      AN    "DI_FW_1".ErrIn.Alarm.NotHalt;
      S     "DI_FW_1".ErrIn.Alarm.Last_UeW_rechts;

      A     "E_WZ_ok_li_1";
      =     "DI_FW_1".ErrIn.Warnung.Wrn_WZ_niO_li_1;

      A     "E_WZ_ok_li_2";
      =     "DI_FW_1".ErrIn.Warnung.Wrn_WZ_niO_li_2;

      A     "E_WZ_ok_li_3";
      =     "DI_FW_1".ErrIn.Warnung.Wrn_WZ_niO_li_3;

      A     "E_WZ_ok_li_4";
      =     "DI_FW_1".ErrIn.Warnung.Wrn_WZ_niO_li_4;

      A     "E_WZ_ok_re_1";
      =     "DI_FW_1".ErrIn.Warnung.Wrn_WZ_niO_re_1;

      A     "E_WZ_ok_re_2";
      =     "DI_FW_1".ErrIn.Warnung.Wrn_WZ_niO_re_2;

      A     "E_WZ_ok_re_3";
      =     "DI_FW_1".ErrIn.Warnung.Wrn_WZ_niO_re_3;

      A     "E_WZ_ok_re_4";
      =     "DI_FW_1".ErrIn.Warnung.Wrn_WZ_niO_re_4;

// Laser Leuze AMS 348i
      CALL  "FC_AMS_304i"
      ( Eingangswert := "ED_PosInc_348i_TW",
        LE_Status    := "EW_Status_348i_TW",
        FW_Nr        := 1,
        Steuerwort   := "AW_Steuer_348i_TW1"
      );

//      CALL  "FC_KorrPos"
//       TW_Nr   :=1
//       IstPos  :="DI_FW_1".ZST.POSITION
//       ErrCount:="DI_FW_1".TMP.ErrCount_Possys
//       Laser_on:="DI_FW_1".IN.Laser_on
//       PosInc  :="DI_FW_1".ZST.PosInc

//  Seillängengeber TR electronic links
      CALL  "FC_IncHub"
      ( Eingangswert      := "ED_HubInc_li_TW",
        Direction         := "DI_FW_1".PAR.Hub.Dir_negativ_li,
        Offset            := "DI_FW_1".PAR.Hub.MessOffset_li,
        Anz_FM            := 5,
        Faktor_Umrechnung := 0.08333334,
        Alarm             := "DI_FW_1".ErrIn.Alarm.HubSys_li,
        count             := "DI_FW_1".PAR.Hub.ErrCount_li,
        Messwert          := "DI_FW_1".ZST.HubInc_li
      );


//Stellung Unten
      L     "DI_FW_1".ZST.HubInc_li;
      L     "DI_FW_1".PAR.Hub.Ebene0;
      -D;
      DTR;
      ABS;
      RND;
      L     "DI_FW_1".PAR.Hub.Bereich_Pos;
      <=D;
      =     "DI_FW_1".IN.Unten_li;

//Stellung oben
      L     "DI_FW_1".ZST.HubInc_li;
      L     "DI_FW_1".PAR.Hub.Ebene3;
      -D;
      DTR;
      ABS;
      RND;
      L     "DI_FW_1".PAR.Hub.Bereich_Pos;
      <=D;
      =     "DI_FW_1".IN.Oben_li;

//  Seillängengeber TR electronic rechts
      CALL  "FC_IncHub"
      ( Eingangswert      := "ED_HubInc_re_TW",
        Direction         := "DI_FW_1".PAR.Hub.Dir_negativ_re,
        Offset            := "DI_FW_1".PAR.Hub.MessOffset_re,
        Anz_FM            := 5,
        Faktor_Umrechnung := 0.08333334,
        Alarm             := "DI_FW_1".ErrIn.Alarm.HubSys_re,
        count             := "DI_FW_1".PAR.Hub.ErrCount_re,
        Messwert          := "DI_FW_1".HELP.HubInc_re
      );

//Stellung Unten
      L     "DI_FW_1".HELP.HubInc_re;
      L     "DI_FW_1".PAR.Hub.Ebene0;
      -D;
      DTR;
      ABS;
      RND;
      L     "DI_FW_1".PAR.Hub.Bereich_Pos;
      <=D;
      =     "DI_FW_1".IN.Unten_re;

//Stellung oben
      L     "DI_FW_1".HELP.HubInc_re;
      L     "DI_FW_1".PAR.Hub.Ebene3;
      -D;
      DTR;
      ABS;
      RND;
      L     "DI_FW_1".PAR.Hub.Bereich_Pos;
      <=D;
      =     "DI_FW_1".IN.Oben_re;


NETWORK
TITLE = Stände / QF
// 6 Be-/Entladepositionen
// 1: vorne links [25]
// 2: vorne rechts [26]
// 3: Großoptiklinks [27]
// 4: Großoptik rechts [28]
// 5: hinten links [29]
// 6: hinten rechts [30]
//Beladestand 1 ------------------------
      AN    "E_S_vl_QF1_frei";
      AN    "E_S_hl_QF1_frei";
      O     "DB_BE_Stand".Langware_vorn;
      AN    "DB_BE_Stand".Stand[3].IN_Belegt;
      =     "DB_BE_Stand".Stand[1].IN_Belegt;

// Eingefahren (Übergabeposition)
      A     "E_S_Pos_Ue_QF1";
      AN    "E_S_Pos_BE_QF1";
      AN    "A_Frg_FU_QF_WR02";
      =     "DB_BE_Stand".Stand[1].IN_innen;

      A     "E_S_Pos_BE_QF1";
      AN    "E_S_Pos_Ue_QF1";
      AN    "A_Frg_FU_QF_WR02";
      =     "DB_BE_Stand".Stand[1].IN_aussen;

      A     "E_S_Pos_Ue_QF1";
      AN    "A_Frg_FU_QF_WR02";
      =     "DB_BE_Stand".Stand[1].verriegelt;

      A     "E_T_Frg_BE";
      FP    "DB_BE_Stand".Stand[1].AM_Freigabe;
      A     "DB_BE_Stand".Stand[1].WT_aufgegeben;
      A     "DB_BE_Stand".Stand[1].IN_aussen;
      =     "DB_BE_Stand".Stand[1].IN_Freigabe;

//Beladestand 2 ------------------------
      AN    "E_S_vr_QF1_frei";
      AN    "E_S_hr_QF1_frei";
      O     "DB_BE_Stand".Langware_vorn;
      AN    "DB_BE_Stand".Stand[4].IN_Belegt;
      =     "DB_BE_Stand".Stand[2].IN_Belegt;

      A     "DB_BE_Stand".Stand[1].IN_innen;
      =     "DB_BE_Stand".Stand[2].IN_innen;

      A     "DB_BE_Stand".Stand[1].IN_aussen;
      =     "DB_BE_Stand".Stand[2].IN_aussen;

      A     "DB_BE_Stand".Stand[1].verriegelt;
      =     "DB_BE_Stand".Stand[2].verriegelt;

      A     "E_T_Frg_BE";
      FP    "DB_BE_Stand".Stand[2].AM_Freigabe;
      A     "DB_BE_Stand".Stand[2].WT_aufgegeben;
      A     "DB_BE_Stand".Stand[2].IN_aussen;
      =     "DB_BE_Stand".Stand[2].IN_Freigabe;

// Anforderung Großoptik via Panel
      A     "Panel".Aufgabe.Anf_GO;
      S     "DI_QF_WR02_03".In.Req_Aufgabe_GO;
      R     "Panel".Aufgabe.Anf_GO;

      A     "DB_BE_Stand".Stand[3].IN_innen;
      A(;
      A     "DB_BE_Stand".Stand[3].WT_aufgegeben;
      O     "DB_BE_Stand".Stand[4].WT_aufgegeben;
      );
      O     "DB_ANLAGE".BA.Tippbetrieb;
      R     "DI_QF_WR02_03".In.Req_Aufgabe_GO;

// Änderung Klingberg 4.1.2024
// Um die Anwahl, ohne größere Änderung, zu Visualisieren,
// wird das Bit auf einen Merker kopiert.
      A     "DI_QF_WR02_03".In.Req_Aufgabe_GO;
      =     "GrossoptikIstAngefordert";

//Beladestand 3 ------------------------
      AN    "E_S_vl_QF1_frei";
      ON    "E_S_hl_QF1_frei";
      ON    "E_S_vl_QF2_frei";
//      ON    "E_S_hl_QF2_frei"
      L     S5T#5s;
      Extend "T_GO_links";

      AN    "E_S_vl_QF1_frei";
      AN    "E_S_hl_QF1_frei";
      AN    "E_S_vl_QF2_frei";
      A     "E_S_hl_QF2_frei";
      A     "T_GO_links";
      S     "DB_BE_Stand".Stand[3].IN_Belegt;

      A     "E_S_vl_QF1_frei";
      A     "E_S_hl_QF1_frei";
      A     "E_S_vl_QF2_frei";
      A     "E_S_hl_QF2_frei";
      R     "DB_BE_Stand".Stand[3].IN_Belegt;

// Eingefahren (Übergabeposition)
      A     "DB_BE_Stand".Stand[1].IN_innen;
      A     "DB_BE_Stand".Stand[5].IN_innen;
      =     "DB_BE_Stand".Stand[3].IN_innen;

      A     "DB_BE_Stand".Stand[1].IN_aussen;
      A     "DB_BE_Stand".Stand[5].IN_aussen;
      =     "DB_BE_Stand".Stand[3].IN_aussen;


      A     "DB_BE_Stand".Stand[1].verriegelt;
      A     "DB_BE_Stand".Stand[5].verriegelt;
      =     "DB_BE_Stand".Stand[3].verriegelt;

      A     "E_T_Frg_BE";
      FP    "DB_BE_Stand".Stand[3].AM_Freigabe;
      A     "DB_BE_Stand".Stand[3].WT_aufgegeben;
      A     "DB_BE_Stand".Stand[3].IN_aussen;
      =     "DB_BE_Stand".Stand[3].IN_Freigabe;

//Beladestand 4 ------------------------
      AN    "E_S_vr_QF1_frei";
      ON    "E_S_hr_QF1_frei";
//      ON    "E_S_vr_QF2_frei"
      ON    "E_S_hr_QF2_frei";
      L     S5T#5s;
      Extend "T_GO_rechts";

      AN    "E_S_vr_QF1_frei";
      AN    "E_S_hr_QF1_frei";
      A     "E_S_vr_QF2_frei";
      AN    "E_S_hr_QF2_frei";
      A     "T_GO_rechts";
      S     "DB_BE_Stand".Stand[4].IN_Belegt;

      A     "E_S_vr_QF1_frei";
      A     "E_S_hr_QF1_frei";
      A     "E_S_vr_QF2_frei";
      A     "E_S_hr_QF2_frei";
      R     "DB_BE_Stand".Stand[4].IN_Belegt;

// Eingefahren (Übergabeposition)
      A     "DB_BE_Stand".Stand[2].IN_innen;
      A     "DB_BE_Stand".Stand[6].IN_innen;
      =     "DB_BE_Stand".Stand[4].IN_innen;

      A     "DB_BE_Stand".Stand[2].IN_aussen;
      A     "DB_BE_Stand".Stand[6].IN_aussen;
      =     "DB_BE_Stand".Stand[4].IN_aussen;

      A     "DB_BE_Stand".Stand[1].verriegelt;
      A     "DB_BE_Stand".Stand[5].verriegelt;
      =     "DB_BE_Stand".Stand[4].verriegelt;

      A     "E_T_Frg_BE";
      FP    "DB_BE_Stand".Stand[4].AM_Freigabe;
      A     "DB_BE_Stand".Stand[4].WT_aufgegeben;
      A     "DB_BE_Stand".Stand[4].IN_aussen;
      =     "DB_BE_Stand".Stand[4].IN_Freigabe;

//Beladestand 5 ------------------------
      AN    "E_S_vl_QF2_frei";
      AN    "E_S_hl_QF2_frei";
      O     "DB_BE_Stand".Langware_hinten;
      AN    "DB_BE_Stand".Stand[3].IN_Belegt;
      =     "DB_BE_Stand".Stand[5].IN_Belegt;

// Eingefahren (Übergabeposition)
      A     "E_S_Pos_Ue_QF2";
      AN    "E_S_Pos_BE_QF2";
      AN    "A_Frg_FU_QF_WR03";
      =     "DB_BE_Stand".Stand[5].IN_innen;

      A     "E_S_Pos_BE_QF2";
      AN    "E_S_Pos_Ue_QF2";
      AN    "A_Frg_FU_QF_WR03";
      =     "DB_BE_Stand".Stand[5].IN_aussen;

      A     "E_S_Pos_Ue_QF2";
      AN    "A_Frg_FU_QF_WR03";
      =     "DB_BE_Stand".Stand[5].verriegelt;

      A     "E_T_Frg_BE";
      FP    "DB_BE_Stand".Stand[5].AM_Freigabe;
      A     "DB_BE_Stand".Stand[5].WT_aufgegeben;
      A     "DB_BE_Stand".Stand[5].IN_aussen;
      =     "DB_BE_Stand".Stand[5].IN_Freigabe;

//Beladestand 6 ------------------------
      AN    "E_S_vr_QF2_frei";
      AN    "E_S_hr_QF2_frei";
      O     "DB_BE_Stand".Langware_hinten;
      AN    "DB_BE_Stand".Stand[4].IN_Belegt;
      =     "DB_BE_Stand".Stand[6].IN_Belegt;

// Eingefahren (Übergabeposition)
      A     "DB_BE_Stand".Stand[5].IN_innen;
      =     "DB_BE_Stand".Stand[6].IN_innen;

      A     "DB_BE_Stand".Stand[5].IN_aussen;
      =     "DB_BE_Stand".Stand[6].IN_aussen;

      A     "DB_BE_Stand".Stand[5].verriegelt;
      =     "DB_BE_Stand".Stand[6].verriegelt;

      A     "E_T_Frg_BE";
      FP    "DB_BE_Stand".Stand[6].AM_Freigabe;
      A     "DB_BE_Stand".Stand[6].WT_aufgegeben;
      A     "DB_BE_Stand".Stand[6].IN_aussen;
      =     "DB_BE_Stand".Stand[6].IN_Freigabe;

// Aufgabe-Button freigen (--> Panel)
      L     "DB_Prog_edit".Prog_Aufgabe.Prog.Geometrie;
      L     #Aufgabe_KS;
      ==I;
      A(;
      L     "DB_Prog_edit".Prog_Aufgabe.Korb_Nr;
      L     0;
      <>I;
      );
      A(;
      L     "DB_Optimierung_HCA".Restzeit_Kurz_Links;
      L     0;
      ==D;
      );
      A     "DB_BE_Stand".Stand[1].Aufgabe_erlaubt;
      AN    "DB_BE_Stand".Langware_vorn;
      A     "DI_FW_Auftrag_DB".Frg_Einfahrt;
      =     "Panel".Aufgabe.KS_vl_erlaubt;

      L     "DB_Prog_edit".Prog_Aufgabe.Prog.Geometrie;
      L     #Aufgabe_KS;
      ==I;
      A(;
      L     "DB_Prog_edit".Prog_Aufgabe.Korb_Nr;
      L     0;
      <>I;
      );
      A(;
      L     "DB_Optimierung_HCA".Restzeit_Kurz_Rechts;
      L     0;
      ==D;
      );
      A     "DB_BE_Stand".Stand[2].Aufgabe_erlaubt;
      AN    "DB_BE_Stand".Langware_vorn;
      A     "DI_FW_Auftrag_DB".Frg_Einfahrt;
      =     "Panel".Aufgabe.KS_vr_erlaubt;

      L     "DB_Prog_edit".Prog_Aufgabe.Prog.Geometrie;
      L     #Aufgabe_GO;
      ==I;
      A(;
      L     "DB_Prog_edit".Prog_Aufgabe.Korb_Nr;
      L     0;
      <>I;
      );
      A(;
      L     "DB_Optimierung_HCA".Restzeit_Gross_Links;
      L     0;
      ==D;
      );
      A     "DB_BE_Stand".Stand[3].Aufgabe_erlaubt;
      A     "DI_FW_Auftrag_DB".Frg_Einfahrt;
      =     "Panel".Aufgabe.GO_li_erlaubt;

      L     "DB_Prog_edit".Prog_Aufgabe.Prog.Geometrie;
      L     #Aufgabe_GO;
      ==I;
      A(;
      L     "DB_Prog_edit".Prog_Aufgabe.Korb_Nr;
      L     0;
      <>I;
      );
      A(;
      L     "DB_Optimierung_HCA".Restzeit_Gross_Rechts;
      L     0;
      ==D;
      );
      A     "DB_BE_Stand".Stand[4].Aufgabe_erlaubt;
      A     "DI_FW_Auftrag_DB".Frg_Einfahrt;
      =     "Panel".Aufgabe.GO_re_erlaubt;

      L     "DB_Prog_edit".Prog_Aufgabe.Prog.Geometrie;
      L     #Aufgabe_KS;
      ==I;
      A(;
      L     "DB_Prog_edit".Prog_Aufgabe.Korb_Nr;
      L     0;
      <>I;
      );
      A(;
      L     "DB_Optimierung_HCA".Restzeit_Kurz_Links;
      L     0;
      ==D;
      );
      A     "DB_BE_Stand".Stand[5].Aufgabe_erlaubt;
      AN    "DB_BE_Stand".Langware_hinten;
      A     "DI_FW_Auftrag_DB".Frg_Einfahrt;
      =     "Panel".Aufgabe.KS_hl_erlaubt;

      L     "DB_Prog_edit".Prog_Aufgabe.Prog.Geometrie;
      L     #Aufgabe_KS;
      ==I;
      A(;
      L     "DB_Prog_edit".Prog_Aufgabe.Korb_Nr;
      L     0;
      <>I;
      );
      A(;
      L     "DB_Optimierung_HCA".Restzeit_Kurz_Rechts;
      L     0;
      ==D;
      );
      A     "DB_BE_Stand".Stand[6].Aufgabe_erlaubt;
      AN    "DB_BE_Stand".Langware_hinten;
      A     "DI_FW_Auftrag_DB".Frg_Einfahrt;
      =     "Panel".Aufgabe.KS_hr_erlaubt;

// Langware vorne
      AN    "E_S_hl_QF1_frei";
      ON    "E_S_hr_QF1_frei";
      L     S5T#5s;
      Extend "T_LS_vorn";

      AN    "E_S_hl_QF1_frei";
      A     "E_S_vl_QF1_frei";
      AN    "E_S_hr_QF1_frei";
      A     "E_S_vr_QF1_frei";
      A     "T_LS_vorn";
      S     "DB_BE_Stand".Langware_vorn;

      L     "DB_Prog_edit".Prog_Aufgabe.Prog.Geometrie;
      L     #Aufgabe_LS;
      ==I;
      A(;
      L     "DB_Prog_edit".Prog_Aufgabe.Korb_Nr;
      L     0;
      <>I;
      );
      A     "DB_BE_Stand".Langware_vorn;
      A     "DB_BE_Stand".Stand[1].Aufgabe_erlaubt;
      A     "DI_FW_Auftrag_DB".Frg_Einfahrt;
      =     "Panel".Aufgabe.LS_v_erlaubt;

      A     "E_S_vl_QF1_frei";
      A     "E_S_hl_QF1_frei";
      A     "E_S_vr_QF1_frei";
      A     "E_S_hr_QF1_frei";
      R     "DB_BE_Stand".Langware_vorn;

// Langware hinten
      AN    "E_S_hl_QF2_frei";
      ON    "E_S_hr_QF2_frei";
      L     S5T#5s;
      Extend "T_LS_hinten";

      AN    "E_S_hl_QF2_frei";
      A     "E_S_vl_QF2_frei";
      AN    "E_S_hr_QF2_frei";
      A     "E_S_vr_QF2_frei";
      A     "T_LS_hinten";
      S     "DB_BE_Stand".Langware_hinten;

      L     "DB_Prog_edit".Prog_Aufgabe.Prog.Geometrie;
      L     #Aufgabe_LS;
      ==I;
      A(;
      L     "DB_Prog_edit".Prog_Aufgabe.Korb_Nr;
      L     0;
      <>I;
      );
      A     "DB_BE_Stand".Langware_hinten;
      A     "DB_BE_Stand".Stand[5].Aufgabe_erlaubt;
      A     "DI_FW_Auftrag_DB".Frg_Einfahrt;
      =     "Panel".Aufgabe.LS_h_erlaubt;

      A     "E_S_vl_QF2_frei";
      A     "E_S_hl_QF2_frei";
      A     "E_S_vr_QF2_frei";
      A     "E_S_hr_QF2_frei";
      R     "DB_BE_Stand".Langware_hinten;

// Fertiganzeige B/E
      A     "DB_POS".POS[25].belegt;
      A     "DB_POS".POS[25].Belegt_KS;
      A     "DB_POS".POS[25].OUTA;
      =     "Panel".QF.P25_kurz_fertig;

      A     "DB_POS".POS[25].belegt;
      A     "DB_POS".POS[25].Belegt_LS;
      A     "DB_POS".POS[25].OUTA;
      =     "Panel".QF.P25_lang_fertig;

      A     "DB_POS".POS[26].belegt;
      A     "DB_POS".POS[26].Belegt_KS;
      A     "DB_POS".POS[26].OUTA;
      =     "Panel".QF.P26_fertig;

      A     "DB_POS".POS[27].belegt;
      A     "DB_POS".POS[27].Belegt_GO;
      A     "DB_POS".POS[27].OUTA;
      =     "Panel".QF.P27_fertig;

      A     "DB_POS".POS[28].belegt;
      A     "DB_POS".POS[28].Belegt_GO;
      A     "DB_POS".POS[28].OUTA;
      =     "Panel".QF.P28_fertig;

      A     "DB_POS".POS[29].belegt;
      A     "DB_POS".POS[29].Belegt_KS;
      A     "DB_POS".POS[29].OUTA;
      =     "Panel".QF.P29_kurz_fertig;

      A     "DB_POS".POS[29].belegt;
      A     "DB_POS".POS[29].Belegt_LS;
      A     "DB_POS".POS[29].OUTA;
      =     "Panel".QF.P29_lang_fertig;

      A     "DB_POS".POS[30].belegt;
      A     "DB_POS".POS[30].Belegt_KS;
      A     "DB_POS".POS[30].OUTA;
      =     "Panel".QF.P30_fertig;

// BA
      A     "DB_ANLAGE".BA.Tippbetrieb;
      =     "DI_QF_WR02_03".In.Tipp;
      A     "DB_ANLAGE".BA.Handbetrieb;
      =     "DI_QF_WR02_03".In.Hand;
      A     "DB_ANLAGE".BA.Automat_ein;
      =     "DI_QF_WR02_03".In.Auto;
// Fehlerquittung
      A     "DB_ANLAGE".IN.Quitt_Err;
      =     "DI_QF_WR02_03".In.ErrQ;

// WR02
// Tasten
      A     "Panel".QF.WR02.T_einfahren;
      =     "DI_QF_WR02_03".In.T_WR02_zu_UE;
      A     "Panel".QF.WR02.T_ausfahren;
      =     "DI_QF_WR02_03".In.T_WR02_zu_BE;

      A     "T_MobielPanel_Lebensbit_ein";
      O     "T_MobielPanel_Lebensbit_aus";
      R     "Panel".QF.WR02.T_einfahren;
      R     "Panel".QF.WR02.T_ausfahren;

// Sensoren
      A     "E_S_Pos_Ue_QF1";
      =     "DI_QF_WR02_03".In.S_WR02_UE;
      A     "E_S_Pos_BE_QF1";
      =     "DI_QF_WR02_03".In.S_WR02_BE;
      A     "E_S_lgsm_to_Ue_QF1";
      =     "DI_QF_WR02_03".In.S_WR02_lgsm_UE;
      A     "E_S_lgsm_to_BE_QF1";
      =     "DI_QF_WR02_03".In.S_WR02_lgsm_BE;

// --> Panel
      A     "DI_QF_WR02_03".In.S_WR02_UE;
      =     "Panel".QF.WR02.S_Pos_Ue;
      A     "DI_QF_WR02_03".In.S_WR02_BE;
      =     "Panel".QF.WR02.S_Pos_BE;
      A     "DI_QF_WR02_03".Out.WR02_einfahren;
      =     "Panel".QF.WR02.A_einfahren;
      A     "DI_QF_WR02_03".Out.WR02_ausfahren;
      =     "Panel".QF.WR02.A_ausfahren;

      AN    "E_S_vl_QF1_frei";
      =     "Panel".QF.WR02.S_BK_vl;
      AN    "E_S_vr_QF1_frei";
      =     "Panel".QF.WR02.S_BK_vr;
      AN    "E_S_hl_QF1_frei";
      =     "Panel".QF.WR02.S_BK_hl;
      AN    "E_S_hr_QF1_frei";
      =     "Panel".QF.WR02.S_BK_hr;

// FU[8] - WR02
      A     "FU_In_Out".FU[8].PE.Statusbyte.Stoer;
      =     "DI_QF_WR02_03".In.FU_Stoerung_WR02;
      A     "FU_In_Out".FU[8].PE.Statusbyte.Bereit;
      =     "DI_QF_WR02_03".In.FU_betriebsbereit_WR02;

//WR03
//Tasten
      A     "Panel".QF.WR03.T_einfahren;
      =     "DI_QF_WR02_03".In.T_WR03_zu_UE;
      A     "Panel".QF.WR03.T_ausfahren;
      =     "DI_QF_WR02_03".In.T_WR03_zu_BE;

      A     "T_MobielPanel_Lebensbit_ein";
      O     "T_MobielPanel_Lebensbit_aus";
      R     "Panel".QF.WR03.T_einfahren;
      R     "Panel".QF.WR03.T_ausfahren;

// Sensoren
      A     "E_S_Pos_Ue_QF2";
      =     "DI_QF_WR02_03".In.S_WR03_UE;
      A     "E_S_Pos_BE_QF2";
      =     "DI_QF_WR02_03".In.S_WR03_BE;

      A     "E_S_lgsm_to_Ue_QF2";
      =     "DI_QF_WR02_03".In.S_WR03_lgsm_UE;
      A     "E_S_lgsm_to_BE_QF2";
      =     "DI_QF_WR02_03".In.S_WR03_lgsm_BE;

// --> Panel
      A     "DI_QF_WR02_03".In.S_WR03_UE;
      =     "Panel".QF.WR03.S_Pos_Ue;
      A     "DI_QF_WR02_03".In.S_WR03_BE;
      =     "Panel".QF.WR03.S_Pos_BE;
      A     "DI_QF_WR02_03".Out.WR03_einfahren;
      =     "Panel".QF.WR03.A_einfahren;
      A     "DI_QF_WR02_03".Out.WR03_ausfahren;
      =     "Panel".QF.WR03.A_ausfahren;

      AN    "E_S_vl_QF2_frei";
      =     "Panel".QF.WR03.S_BK_vl;
      AN    "E_S_vr_QF2_frei";
      =     "Panel".QF.WR03.S_BK_vr;
      AN    "E_S_hl_QF2_frei";
      =     "Panel".QF.WR03.S_BK_hl;
      AN    "E_S_hr_QF2_frei";
      =     "Panel".QF.WR03.S_BK_hr;

// FU[9] - WR03
      A     "FU_In_Out".FU[9].PE.Statusbyte.Stoer;
      =     "DI_QF_WR02_03".In.FU_Stoerung_WR03;
      A     "FU_In_Out".FU[9].PE.Statusbyte.Bereit;
      =     "DI_QF_WR02_03".In.FU_betriebsbereit_WR03;



NETWORK
TITLE = Dosierung
// 8 Dosierpumpen
// DP1 Verwerfen CM01 (WT)
      A     "E_Imp_GP02.BF02";
      A     "DB_DP".DP[1].Dosi_akt;
      AN    "DB_DP".DP[1].DP_OFF;
      =     "DB_DP".DP[1].DP_Imp;
// DP2 Nachschärfen CM01 (WT)
      A     "E_Imp_GP01.BF01";
      A     "DB_DP".DP[2].Dosi_akt;
      AN    "DB_DP".DP[2].DP_OFF;
      =     "DB_DP".DP[2].DP_Imp;

// DP3 Verwerfen CM02 (WT)
      A     "E_Imp_GP02.BF02";
      A     "DB_DP".DP[3].Dosi_akt;
      AN    "DB_DP".DP[3].DP_OFF;
      =     "DB_DP".DP[3].DP_Imp;
// DP4 Nachschärfen CM02 (WT)
      A     "E_Imp_GP01.BF01";
      A     "DB_DP".DP[4].Dosi_akt;
      AN    "DB_DP".DP[4].DP_OFF;
      =     "DB_DP".DP[4].DP_Imp;

// Optional
// DP5 Verwerfen CM01 (LF)
      A     "E_Imp_GP02.BF02";
      A     "DB_DP".DP[5].Dosi_akt;
      AN    "DB_DP".DP[5].DP_OFF;
      =     "DB_DP".DP[5].DP_Imp;
// DP6 Nachschärfen CM01(LF)
      A     "E_Imp_GP01.BF01";
      A     "DB_DP".DP[6].Dosi_akt;
      AN    "DB_DP".DP[6].DP_OFF;
      =     "DB_DP".DP[6].DP_Imp;

// DP7 Verwerfen CM02 (LF)
      A     "E_Imp_GP02.BF02";
      A     "DB_DP".DP[7].Dosi_akt;
      AN    "DB_DP".DP[7].DP_OFF;
      =     "DB_DP".DP[7].DP_Imp;
// DP8 Nachschärfen CM02 (LF)
      A     "E_Imp_GP01.BF01";
      A     "DB_DP".DP[8].Dosi_akt;
      AN    "DB_DP".DP[8].DP_OFF;
      =     "DB_DP".DP[8].DP_Imp;


NETWORK
TITLE = Peripherie
// Eingäne / Panel einlesen
      CALL  "Input_Peripherie";

NETWORK
TITLE = Deckelsperren
// CM01
      SET;
      R     "DB_POS".POS[1].Sperre_FW;
      R     "DB_POS".POS[2].Sperre_FW;
      R     "DB_POS".POS[3].Sperre_FW;
      R     "DB_POS".POS[4].Sperre_FW;
      R     "DB_POS".POS[5].Sperre_FW;
      R     "DB_POS".POS[6].Sperre_FW;

      A     "Deckel_CM01".Zst.Sperre_Pos_li;
      O     "Deckel_CM01".Zst.Sperre_Pos_re;
      =     "DB_Sperrbereiche".Bereich[1].aktiv;

      A(;
      A     "Deckel_CM01".Zst.Req_links_auf;
      AN    "Deckel_CM01".In.S_links_auf;
      O;
      A     "Deckel_CM01".Zst.Req_rechts_auf;
      AN    "Deckel_CM01".In.S_rechts_auf;
      );
      A     "Deckel_CM01".Zst.TW_sicher;
      S     "DB_Sperrbereiche".Bereich[1].aktiv;

// TW oben und nicht Schmalware
      A     "DI_FW_1".ZST.Oben_li;
      =     "DB_Sperrbereiche".Sperre_links;
      A     "DI_FW_1".ZST.Oben_re;
      =     "DB_Sperrbereiche".Sperre_rechts;

      L     0;
      L     "DI_FW_1".ZST.WT_DB_NR_li;
      >=I;
      JC    Chre;
      +     100;
      T     #WT_DB;
      OPN   DB [#WT_DB];
      L     "WT_Typ_KS";
      L     %DBB35;
      ==I;
      O(;
      L     "WT_Typ_LS";
      ==I;
      );
      R     "DB_Sperrbereiche".Sperre_links;

Chre: L     0;
      L     "DI_FW_1".ZST.WT_DB_NR_re;
      >=I;
      JC    s_SP;
      +     100;
      T     #WT_DB;
      OPN   DB [#WT_DB];
      L     "WT_Typ_KS";
      L     %DBB35;
      ==I;
      O(;
      L     "WT_Typ_LS";
      ==I;
      );
      R     "DB_Sperrbereiche".Sperre_rechts;

s_SP: A     "DB_Sperrbereiche".Sperre_links;
      O     "DB_Sperrbereiche".Sperre_rechts;
      A     "DB_Sperrbereiche".Bereich[1].aktiv;
      =     "DB_Sperrbereiche".Bereich[3].aktiv;

      AN    "Deckel_CM01".In.S_links_auf;
      O     "Deckel_CM01".Zst.Sperre_Pos_li;
      =     "DB_POS".POS[1].IN_OUT_nen;
      =     "DB_POS".POS[3].IN_OUT_nen;
      =     "DB_POS".POS[5].IN_OUT_nen;

      AN    "Deckel_CM01".In.S_rechts_auf;
      O     "Deckel_CM01".Zst.Sperre_Pos_re;
      =     "DB_POS".POS[2].IN_OUT_nen;
      =     "DB_POS".POS[4].IN_OUT_nen;
      =     "DB_POS".POS[6].IN_OUT_nen;

// CM02
      SET;
      R     "DB_POS".POS[13].Sperre_FW;
      R     "DB_POS".POS[14].Sperre_FW;
      R     "DB_POS".POS[15].Sperre_FW;
      R     "DB_POS".POS[16].Sperre_FW;
      R     "DB_POS".POS[17].Sperre_FW;
      R     "DB_POS".POS[18].Sperre_FW;

      A     "Deckel_CM02".Zst.Sperre_Pos_li;
      O     "Deckel_CM02".Zst.Sperre_Pos_re;
      =     "DB_Sperrbereiche".Bereich[2].aktiv;

      A(;
      A     "Deckel_CM02".Zst.Req_links_auf;
      AN    "Deckel_CM02".In.S_links_auf;
      O;
      A     "Deckel_CM02".Zst.Req_rechts_auf;
      AN    "Deckel_CM02".In.S_rechts_auf;
      );
      A     "Deckel_CM02".Zst.TW_sicher;
      S     "DB_Sperrbereiche".Bereich[2].aktiv;


      A     "DB_Sperrbereiche".Sperre_links;
      O     "DB_Sperrbereiche".Sperre_rechts;
      A     "DB_Sperrbereiche".Bereich[2].aktiv;
      =     "DB_Sperrbereiche".Bereich[4].aktiv;

      AN    "Deckel_CM02".In.S_links_auf;
      O     "Deckel_CM02".Zst.Sperre_Pos_li;
      =     "DB_POS".POS[13].IN_OUT_nen;
      =     "DB_POS".POS[15].IN_OUT_nen;
      =     "DB_POS".POS[17].IN_OUT_nen;

      AN    "Deckel_CM02".In.S_rechts_auf;
      O     "Deckel_CM02".Zst.Sperre_Pos_re;
      =     "DB_POS".POS[14].IN_OUT_nen;
      =     "DB_POS".POS[16].IN_OUT_nen;
      =     "DB_POS".POS[18].IN_OUT_nen;

// Abstand rückwärts Querförderer umschalten
      A     "DB_Sperrbereiche".Sperre_links;
      O     "DB_Sperrbereiche".Sperre_rechts;
      L     1595;  // Abstand für Großoptik
      JC    SpGO;
      L     1029;  // "normal"
SpGO: T     "DB_POS".POS[25].IncAbstand_rck;

END_FUNCTION

FUNCTION "FC_AMS_304i" : Void   // FC204, STL
TITLE = Absolut-Wegmessung
{ S7_Optimized_Access := 'FALSE' }
// stored: AutoNumber false
   VAR_INPUT
      Eingangswert : DInt;   // kompletter Eingangswert
      LE_Status : Word;   // Status enthält Diodenstatus und Fehler vom Gerät
      FW_Nr : Int;   // Fahrwagen-Nr.
   END_VAR
   VAR_IN_OUT
      Steuerwort : Word;   // Laserdiode ein-/ausschalten
   END_VAR
   VAR_TEMP
      Messung : DInt;   // neuer gemessener Wert
      Messwert : DInt;   // Messwert in mm
      Offset : DInt;
      DB_Nr : Word;
      FW_DB : Word;
      count : Byte;
      Req_Laser : Bool;   // Anforderung Messwert
      invers : Bool;
      Laser_on : Bool;
      Alarm : Bool;
      Warng_Signal : Bool;
      Warng_Temp : Bool;
      Warng_Plausi : Bool;
      Anz_FM : Int;   // Anzahl Fehlmessungen
      Laser_was_on : Bool;
   END_VAR
BEGIN

NETWORK
TITLE = Werte aus FW holen
//----------------------------
// Aufbereitung Eingangswerte
//----------------------------
      L     #FW_Nr;
      L     10;
      +I;
      T     #FW_DB;
      OPN   DB [#FW_DB];
      L     0;
      L     %DBB210;  //"DI_FW_1".PAR.Fahrt.Dir_negativ
      <>I;
      =     #invers;

      L     %DBD206;  //"DI_FW_1".PAR.Fahrt.MessOffset
      T     #Offset;

      A     %DBX70.3;  //"DI_FW_1".OUT.Req_Laser
      =     #Req_Laser;

      A     %DBX51.7;  //"DI_FW_1".IN.Laser_on
      =     #Laser_on;

      L     %DBB211;  //"DI_FW_1".PAR.Fahrt.ErrCount
      T     #Anz_FM;

      L     %DBB361;  //"DI_FW_1".TMP.ErrCount_Possys
      T     #count;

      L     %DBD4;  //"DI_FW_1".ZST.PosInc
      T     #Messwert;


NETWORK
TITLE = 
//----------------------
//Warnungen
//----------------------

      A     #Req_Laser;
      AN    #LE_Status.%X0;  //Laser_off
      AN    #LE_Status.%X4;  //Lasersignal zu gering
      S     #Laser_on;

      AN    #Req_Laser;
      R     #Laser_on;

      A     #LE_Status.%X4;  //Lasersignal zu gering
      A     #Laser_on;
      =     #Warng_Signal;  //Signalpegel zu gering

      A     #LE_Status.%X5;  //Temperatur zu hoch
      =     #Warng_Temp;  //Temperatur zu hoch

      A     #LE_Status.%X7;  //Plausibilität
      A     #Laser_on;
      =     #Warng_Plausi;

      A     #LE_Status.%X4;  //Lasersignal zu gering//
      A     #Laser_on;
      =     #Alarm;

      A     #LE_Status.%X8;  //Harwarefehler
      S     #Alarm;

//----------------------
//Laserdiode steuern
//----------------------
      A     #Req_Laser;
      L     0;
      JC    Las;
      L     16#0100;
Las:  T     #Steuerwort;

//----------------------
//Gerät defekt
//----------------------
      A     #Alarm;
      JC    out;

//----------------------
//Laserdiode aus
//----------------------
      A     #Req_Laser;  //neu falls Diode nicht einschaltet
      O     #Laser_on;
      JC    mess;
      L     0;
      T     #count;
      JU    out;
//-----------------
//    Messwert
//-----------------
mess: L     #Eingangswert;
      T     #Messung;
      L     0;
      >D;
      JC    ok;

      L     #Anz_FM;
      A     #Laser_on;
      JC    chk;
      L     2;
      *I;
chk:  L     #count;
      <=I;
      JC    err;
      +     1;
      T     #count;
      JU    out;
err:  SET;
      S     #Alarm;
      JU    out;

ok:   SET;
      R     #Alarm;

      L     0;
      T     #count;

      L     #Offset;
      L     #Messung;
      A     #invers;
      JC    sub;
      +D;
      T     #Messwert;
      JU    out;

sub:  -D;
      T     #Messwert;
      JU    out;


NETWORK
TITLE = 
out:  OPN   DB [#FW_DB];
      L     #count;
      T     %DBB361;  //"DI_FW_1".TMP.ErrCount_Possys

      L     #Messwert;
      T     %DBD4;  //"DI_FW_1".ZST.PosInc

      A     #Warng_Signal;
      =     %DBX66.0;  //"DI_FW_1".ErrIn.Warnung.Wrn_Optik_PosSys
      A     #Warng_Temp;
      =     %DBX66.1;  //"DI_FW_1".ErrIn.Warnung.Wrn_Temp_PosSys
      A     #Warng_Plausi;
      =     %DBX66.2;  //"DI_FW_1".ErrIn.Warnung.Wrn_Plaus_PosSys
      A     #Alarm;
      =     %DBX62.1;  //"DI_FW_1".ErrIn.Alarm.PosSys
      A     #Laser_on;
      =     %DBX51.7;  //"DI_FW_1".IN.Laser_on

END_FUNCTION

FUNCTION "FC_IncHub" : Void   // FC208, STL
TITLE = Absolut-Wegmessung Hub
{ S7_Optimized_Access := 'FALSE' }
// stored: AutoNumber false
   VAR_INPUT
      Eingangswert : DInt;   // kompletter Eingangswert
      Direction : Byte;
      Offset : DInt;
      Anz_FM : Int;   // Anzahl Fehlmessungen
      Faktor_Umrechnung : Real;   // Umrechnung in mm
   END_VAR
   VAR_IN_OUT
      Alarm : Bool;
      count : Byte;
      Messwert : DInt;   // Messwert in mm
   END_VAR
   VAR_TEMP
      Messung : DInt;   // neuer gemessener Wert
      invers : Bool;
   END_VAR
BEGIN

NETWORK
TITLE = 
//-----------------
//    Messwert
//-----------------
      L     0;
      L     #Direction;
      <>I;
      =     #invers;

      L     #Eingangswert;
      T     #Messung;
      L     0;
      <>D;
      JC    ok;

      L     #Anz_FM;
      L     #count;
      <=I;
      JC    err;
      +     1;
      T     #count;
      BE;
err:  SET;
      S     #Alarm;
      BE;

ok:   SET;
      R     #Alarm;

      L     0;
      T     #count;

      L     #Messung;
      AN    #invers;
      JC    sub;
      INVD;
sub:  DTR;
      L     #Faktor_Umrechnung;
      *R;
      RND;
      L     #Offset;
      +D;
      T     #Messwert;
      BE;

END_FUNCTION

FUNCTION "Input_Peripherie" : Void   // FC1010, LAD
TITLE = Input
{ S7_Optimized_Access := 'TRUE' }
// stored: AutoNumber false, SetENOAutomatically true
   VAR_TEMP
      Sperre_Inc_max : DInt;
      Sperre_Inc_min : DInt;
   END_VAR
BEGIN

REGION Network 1 (SCL): Schnelllauftor
   // Motorschutzschalter
   "Tor".In.MSS_ok := "E_MSS_ok_RT";
   // betriebsbereit
   "Tor".In.ok := "E_RT_ok";
   // Paneltasten
   "Tor".In.Knauf_Auto := "DB_ANLAGE".BA.Automat_ein;
   "Tor".In.T_auf := "Panel".RT.T_auf;
   "Tor".In.T_zu := "Panel".RT.T_zu;
   // Sensoren
   "Tor".In.S_auf := "E_S_RT_auf";
   "Tor".In.S_zu := "E_S_RT_zu";
   // --> Panel
   "Panel".RT.MSS_ok := "Tor".In.MSS_ok;
   "Panel".RT.ok := "Tor".In.ok;
   "Panel".RT.S_offen := "Tor".In.S_auf;
   "Panel".RT.S_geschlossen := "Tor".In.S_zu;
   // Automatik
   "Tor".In.Knauf_Auto := "DB_ANLAGE".BA.Automat_ein;
   // Fehlerquittung
   "Tor".In.ErrQ := "DB_ANLAGE".IN.Quitt_Err;
END_REGION

REGION Network 2 (SCL): Deckel
   REGION CM01
       // Sicherungen
       "Deckel_CM01".In.Si_24VDC_links := "E_Si_24VDC_CM01.MM01";
       "Deckel_CM01".In.Si_24VDC_rechts := "E_Si_24VDC_CM01.MM02";
       // Stellrückmeldungen
       "Deckel_CM01".In.SRM_links_auf := "E_Dkl_li_auf_CM01";
       "Deckel_CM01".In.SRM_links_zu := "E_Dkl_li_zu_CM01";
       "Deckel_CM01".In.SRM_rechts_auf := "E_Dkl_re_auf_CM01";
       "Deckel_CM01".In.SRM_rechts_zu := "E_Dkl_re_zu_CM01";
       // Sensoren
       "Deckel_CM01".In.S_links_auf := "E_S_Dkl_li_auf_CM01.BG01" AND NOT "E_S_Dkl_li_zu_CM01.BG02";
       "Deckel_CM01".In.S_links_zu := "E_S_Dkl_li_zu_CM01.BG02" AND NOT "E_S_Dkl_li_auf_CM01.BG01";
       "Deckel_CM01".In.S_rechts_auf := "E_S_Dkl_re_auf_CM01.BG03" AND NOT "E_S_Dkl_re_zu_CM01.BG04";
       "Deckel_CM01".In.S_rechts_zu := "E_S_Dkl_re_zu_CM01.BG04" AND NOT "E_S_Dkl_re_auf_CM01.BG03";
       // Bedienung via Panel
       "Deckel_CM01".In.Auto := "Panel".Deckel.CM01.Auto;
       "Deckel_CM01".In.Hand := "Panel".Deckel.CM01.Hand;
       "Deckel_CM01".In.Tipp := "Panel".Deckel.CM01.Tipp;

       "Deckel_CM01".In.T_links_auf := "Panel".Deckel.CM01.links_auf;
       "Deckel_CM01".In.T_links_zu := "Panel".Deckel.CM01.links_zu;
       "Deckel_CM01".In.T_rechts_auf := "Panel".Deckel.CM01.rechts_auf;
       "Deckel_CM01".In.T_rechts_zu := "Panel".Deckel.CM01.rechts_zu;
       // --> Panel
       "Panel".Deckel.CM01.SRM_links_auf := "Deckel_CM01".In.SRM_links_auf;
       "Panel".Deckel.CM01.SRM_links_zu := "Deckel_CM01".In.SRM_links_zu;
       "Panel".Deckel.CM01.SRM_rechts_auf := "Deckel_CM01".In.SRM_rechts_auf;
       "Panel".Deckel.CM01.SRM_rechts_zu := "Deckel_CM01".In.SRM_rechts_zu;
       "Panel".Deckel.CM01.S_links_auf := "Deckel_CM01".In.S_links_auf;
       "Panel".Deckel.CM01.S_links_zu := "Deckel_CM01".In.S_links_zu;
       "Panel".Deckel.CM01.S_rechts_auf := "Deckel_CM01".In.S_rechts_auf;
       "Panel".Deckel.CM01.S_rechts_zu := "Deckel_CM01".In.S_rechts_zu;
       "Panel".Deckel.CM01.Ist_Pos_links := "Deckel_CM01".Zst.Ist_Pos_links;
       "Panel".Deckel.CM01.Ist_Pos_rechts := "Deckel_CM01".Zst.Ist_Pos_rechts;

       // Transportwagen im sicheren Bereich
       IF "DB_Sperrbereiche".Sperre_links OR "DB_Sperrbereiche".Sperre_rechts THEN
           IF "DI_FW_1".OUT.VOR THEN
               "Deckel_CM01".Zst.TW_sicher := "DI_FW_1".ZST.PosInc >= ("DB_Sperrbereiche".Bereich[3].max_Inc + "DI_FW_1".PAR.Fahrt.Bereich_Pos);
           ELSE
               "Deckel_CM01".Zst.TW_sicher := "DI_FW_1".ZST.PosInc >= ("DB_Sperrbereiche".Bereich[3].max_Inc + "DI_FW_1".PAR.Fahrt.Bereich_lngsm);
           END_IF;
       ELSIF "DI_FW_1".OUT.VOR THEN
           "Deckel_CM01".Zst.TW_sicher := "DI_FW_1".ZST.PosInc >= ("DB_Sperrbereiche".Bereich[1].max_Inc + "DI_FW_1".PAR.Fahrt.Bereich_Pos);
       ELSE
           "Deckel_CM01".Zst.TW_sicher := "DI_FW_1".ZST.PosInc >= ("DB_Sperrbereiche".Bereich[1].max_Inc + "DI_FW_1".PAR.Fahrt.Bereich_lngsm);
       END_IF;

       // Fehlerquittung
       "Deckel_CM01".In.ErrQ := "DB_ANLAGE".IN.Quitt_Err;
   END_REGION ;
   REGION CM02
       // Sicherungen
       "Deckel_CM02".In.Si_24VDC_links := "E_Si_24VDC_CM02.MM03";
       "Deckel_CM02".In.Si_24VDC_rechts := "E_Si_24VDC_CM02.MM04";
       // Stellrückmeldungen
       "Deckel_CM02".In.SRM_links_auf := "E_Dkl_li_auf_CM02";
       "Deckel_CM02".In.SRM_links_zu := "E_Dkl_li_zu_CM02";
       "Deckel_CM02".In.SRM_rechts_auf := "E_Dkl_re_auf_CM02";
       "Deckel_CM02".In.SRM_rechts_zu := "E_Dkl_re_zu_CM02";
       // Sensoren
       "Deckel_CM02".In.S_links_auf := "E_S_Dkl_li_auf_CM02.BG12" AND NOT "E_S_Dkl_li_zu_CM02.BG13";
       "Deckel_CM02".In.S_links_zu := "E_S_Dkl_li_zu_CM02.BG13" AND NOT "E_S_Dkl_li_auf_CM02.BG12";
       "Deckel_CM02".In.S_rechts_auf := "E_S_Dkl_re_auf_CM02.BG14" AND NOT "E_S_Dkl_re_zu_CM02.BG15";
       "Deckel_CM02".In.S_rechts_zu := "E_S_Dkl_re_zu_CM02.BG15" AND NOT "E_S_Dkl_re_auf_CM02.BG14";
       // Bedienung via Panel
       "Deckel_CM02".In.Auto := "Panel".Deckel.CM02.Auto;
       "Deckel_CM02".In.Hand := "Panel".Deckel.CM02.Hand;
       "Deckel_CM02".In.Tipp := "Panel".Deckel.CM02.Tipp;

       "Deckel_CM02".In.T_links_auf := "Panel".Deckel.CM02.links_auf;
       "Deckel_CM02".In.T_links_zu := "Panel".Deckel.CM02.links_zu;
       "Deckel_CM02".In.T_rechts_auf := "Panel".Deckel.CM02.rechts_auf;
       "Deckel_CM02".In.T_rechts_zu := "Panel".Deckel.CM02.rechts_zu;
       // --> Panel
       "Panel".Deckel.CM02.SRM_links_auf := "Deckel_CM02".In.SRM_links_auf;
       "Panel".Deckel.CM02.SRM_links_zu := "Deckel_CM02".In.SRM_links_zu;
       "Panel".Deckel.CM02.SRM_rechts_auf := "Deckel_CM02".In.SRM_rechts_auf;
       "Panel".Deckel.CM02.SRM_rechts_zu := "Deckel_CM02".In.SRM_rechts_zu;
       "Panel".Deckel.CM02.S_links_auf := "Deckel_CM02".In.S_links_auf;
       "Panel".Deckel.CM02.S_links_zu := "Deckel_CM02".In.S_links_zu;
       "Panel".Deckel.CM02.S_rechts_auf := "Deckel_CM02".In.S_rechts_auf;
       "Panel".Deckel.CM02.S_rechts_zu := "Deckel_CM02".In.S_rechts_zu;
       "Panel".Deckel.CM02.Ist_Pos_links := "Deckel_CM02".Zst.Ist_Pos_links;
       "Panel".Deckel.CM02.Ist_Pos_rechts := "Deckel_CM02".Zst.Ist_Pos_rechts;

       // Transportwagen im sicheren Bereich
       IF "DB_Sperrbereiche".Sperre_links OR "DB_Sperrbereiche".Sperre_rechts THEN

           IF "DI_FW_1".OUT.VOR THEN
               "Deckel_CM02".Zst.TW_sicher :=
               ("DI_FW_1".ZST.PosInc <= ("DB_Sperrbereiche".Bereich[4].min_Inc - "DI_FW_1".PAR.Fahrt.Bereich_lngsm)) OR
               ("DI_FW_1".ZST.PosInc >= ("DB_Sperrbereiche".Bereich[4].max_Inc + "DI_FW_1".PAR.Fahrt.Bereich_Pos));

           ELSIF "DI_FW_1".OUT.RUECK THEN
               "Deckel_CM02".Zst.TW_sicher :=
               ("DI_FW_1".ZST.PosInc <= ("DB_Sperrbereiche".Bereich[4].min_Inc - "DI_FW_1".PAR.Fahrt.Bereich_Pos)) OR
               ("DI_FW_1".ZST.PosInc >= ("DB_Sperrbereiche".Bereich[4].max_Inc + "DI_FW_1".PAR.Fahrt.Bereich_lngsm));
           ELSE
               "Deckel_CM02".Zst.TW_sicher :=
               ("DI_FW_1".ZST.PosInc <= ("DB_Sperrbereiche".Bereich[4].min_Inc)) OR
               ("DI_FW_1".ZST.PosInc >= ("DB_Sperrbereiche".Bereich[4].max_Inc));
           END_IF;

       ELSIF "DI_FW_1".OUT.VOR THEN
           "Deckel_CM02".Zst.TW_sicher :=
           ("DI_FW_1".ZST.PosInc <= ("DB_Sperrbereiche".Bereich[2].min_Inc - "DI_FW_1".PAR.Fahrt.Bereich_lngsm)) OR
           ("DI_FW_1".ZST.PosInc >= ("DB_Sperrbereiche".Bereich[2].max_Inc + "DI_FW_1".PAR.Fahrt.Bereich_Pos));

       ELSIF "DI_FW_1".OUT.RUECK THEN
           "Deckel_CM02".Zst.TW_sicher :=
           ("DI_FW_1".ZST.PosInc <= ("DB_Sperrbereiche".Bereich[2].min_Inc - "DI_FW_1".PAR.Fahrt.Bereich_Pos)) OR
           ("DI_FW_1".ZST.PosInc >= ("DB_Sperrbereiche".Bereich[2].max_Inc + "DI_FW_1".PAR.Fahrt.Bereich_lngsm));

       ELSE
           "Deckel_CM02".Zst.TW_sicher :=
           ("DI_FW_1".ZST.PosInc <= ("DB_Sperrbereiche".Bereich[2].min_Inc)) OR
           ("DI_FW_1".ZST.PosInc >= ("DB_Sperrbereiche".Bereich[2].max_Inc));
       END_IF;

       // Fehlerquittung
       "Deckel_CM02".In.ErrQ := "DB_ANLAGE".IN.Quitt_Err;
   END_REGION ;
END_REGION

REGION Network 3 (SCL): CM01
   REGION Filtern
       "FP_CM01.GP01".Param.Name_Pumpe := 'FP_CM01.GP01';
       "FP_CM01.GP01".Param.Name_Filter := 'Filter HQ1';
       // Niveaus
       "FP_CM01.GP01".In.Niv_TLS := "E_Niv_TLS_CM01.BL04";
       "FP_CM01.GP01".In.Niv_min := "E_Niv_Min_CM01.BL03";
       "FP_CM01.GP01".In.Niv_max := "E_Niv_Max_CM01.BL02";
       "FP_CM01.GP01".In.Niv_Uel := NOT "E_Niv_UeL_CM01.BL01";
       "FP_CM01.GP01".In.Frg_Niv_CM05 := NOT "Pu_CM05.GP11_DB".In."Niv_max_CM05.BL01" AND NOT "Pu_CM05.GP11_DB".In."Niv_Uel_CM05.BL05";
       "FP_CM01.GP01".In.Leckage_ok := "E_LS_HQ0x.BL12";
       "FP_CM01.GP01".In.ext_Freigabe := "E_Al_Gas_ok" AND NOT "E_Not-Strom";
       // Ist-Druck Pumpe
       "FP_CM01.GP01".In.Druck_Pumpe := "Panel".IW."p_CM01.BP03";
       // Differenz-Druck Filter
       "FP_CM01.GP01".In.Delta_p_Filter := "Panel".IW."p_HQ01.BP01";

       //Stellrückmeldungen (Filtern)
       "FP_CM01.GP01".In.SRM_Saugseite_auf := "E_SRM_CM01.QM18_auf" AND NOT "E_SRM_CM01.QM18_zu";
       "FP_CM01.GP01".In.SRM_Saugseite_zu := "E_SRM_CM01.QM18_zu" AND NOT "E_SRM_CM01.QM18_auf";
       "FP_CM01.GP01".In.SRM_Eingang_Filter_auf := "E_SRM_HQ01.QM21_auf" AND NOT "E_SRM_HQ01.QM21_zu";
       "FP_CM01.GP01".In.SRM_Eingang_Filter_zu := "E_SRM_HQ01.QM21_zu" AND NOT "E_SRM_HQ01.QM21_auf";
       "FP_CM01.GP01".In.SRM_Ausgang_Filter_auf := "E_SRM_HQ01.QM23_auf" AND NOT "E_SRM_HQ01.QM23_zu";
       "FP_CM01.GP01".In.SRM_Ausgang_Filter_zu := "E_SRM_HQ01.QM23_zu" AND NOT "E_SRM_HQ01.QM23_auf";

       "FP_CM01.GP01".In.SRM_Eingang_Spülltg_P_auf := "E_SRM_CM01.QM19_auf" AND NOT "E_SRM_CM01.QM19_zu";
       "FP_CM01.GP01".In.SRM_Eingang_Spülltg_P_zu := "E_SRM_CM01.QM19_zu" AND NOT "E_SRM_CM01.QM19_auf";
       "FP_CM01.GP01".In.SRM_Eingang_Spülltg_F_auf := "E_SRM_HQ01.QM22_auf" AND NOT "E_SRM_HQ01.QM22_zu";
       "FP_CM01.GP01".In.SRM_Eingang_Spülltg_F_zu := "E_SRM_HQ01.QM22_zu" AND NOT "E_SRM_HQ01.QM22_auf";
       "FP_CM01.GP01".In.SRM_Ausgang_Spülltg_auf := "E_SRM_HQ01.QM24_auf" AND NOT "E_SRM_HQ01.QM24_zu";
       "FP_CM01.GP01".In.SRM_Ausgang_Spülltg_zu := "E_SRM_HQ01.QM24_zu" AND NOT "E_SRM_HQ01.QM24_auf";
       "FP_CM01.GP01".In.SRM_Entluften_auf := "E_SRM_HQ01.LV01_auf" AND NOT "E_SRM_HQ01.LV01_zu";
       "FP_CM01.GP01".In.SRM_Entlueften_zu := "E_SRM_HQ01.LV01_zu" AND NOT "E_SRM_HQ01.LV01_auf";

       // Filtergehäuse
       "FP_CM01.GP01".In.GW_p_FG := "E_GW_p_HQ01.BP01";
       "FP_CM01.GP01".In.Sensor_FG_links := "E_S_FG_li_HQ01.BG07";
       "FP_CM01.GP01".In.Sensor_FG_rechts := "E_S_FG_re_HQ01.BG08";
       "FP_CM01.GP01".In.Einhausung_HQ0x_zu := "DB_PNOZ_IN_Out".In.FG_zu_HQ01;
       "FP_CM01.GP01".Param.WarnGr_FW := "Panel".HQ01.WarnGr_FW;
       "FP_CM01.GP01".Param.Wechsel_FW := "Panel".HQ01.Wechsel_FW;

       // Not-Halt
       "FP_CM01.GP01".In.NotHalt := NOT "DB_PNOZ_IN_Out".In.NH_Frg_FP_CM01;

       "FP_CM01.GP01".In.GW_p_FP := "E_GW_p_CM01.BP03";
       "FP_CM01.GP01".In.GW_LF_FP := "E_GW_LF_CM01.BN01";

       // Frequenzumrichter [Index 1] 
       "FP_CM01.GP01".In.FU_speed := "FU_In_Out".FU[1].PE.Speed;
       "FP_CM01.GP01".In.FU_betriebsbereit := "FU_In_Out".FU[1].PE.Statusbyte.Bereit;
       "FP_CM01.GP01".In.FU_Stoerung := "FU_In_Out".FU[1].PE.Statusbyte.Stoer;
       "FP_CM01.GP01".Param.SW_Hand := "Panel".FP_CM01.SW_Hand;
       "FP_CM01.GP01".Param.SW_Auto_AZ := "Panel".FP_CM01.SW_Auto_AZ;
       "FP_CM01.GP01".Param.SW_Auto_aAZ := "Panel".FP_CM01.SW_Auto_aAZ;

       // Hand
       "FP_CM01.GP01".In.Ein := "Panel".FP_CM01.Ein;
       // Auto
       "FP_CM01.GP01".In.Auto := "Panel".FP_CM01.Auto;
       // Betriebsart
       "FP_CM01.GP01".In.Betriebsart := "Panel".FP_CM01.BA;
       // Spülzeit
       "FP_CM01.GP01".Param.Spülzeit_Pumpe := DINT_TO_TIME(INT_TO_DINT("Panel".FP_CM01.Sp_Ventil.Sollzeit) * 1000);
       // Zeiten Filterwechsel
       "FP_CM01.GP01".Param.FG_Zeit_leeren_Saurebecken := DINT_TO_TIME(INT_TO_DINT("Panel".FP_CM01.Sp_Filter.Zeit_leeren_Saure) * 1000);
       "FP_CM01.GP01".Param.FG_Zeit_leeren_CM05 := DINT_TO_TIME(INT_TO_DINT("Panel".FP_CM01.Sp_Filter.Zeit_leeren_CM05) * 1000);
       "FP_CM01.GP01".Param.FW_Spülzeit := DINT_TO_TIME(INT_TO_DINT("Panel".FP_CM01.Sp_Filter.Zeit_Spülen) * 1000);
       "FP_CM01.GP01".Param.FW_Wartezeit := DINT_TO_TIME(INT_TO_DINT("Panel".FP_CM01.Sp_Filter.Wartezeit) * 1000);
       "FP_CM01.GP01".Param.FW_Zeit_fuellen := DINT_TO_TIME(INT_TO_DINT("Panel".FP_CM01.Sp_Filter.Zeit_füllen) * 1000);
       // Drucktest Pumpe
       "FP_CM01.GP01".Param.DT_Druckaufbau := T#1m;
       "FP_CM01.GP01".Param.SW_Drucktest_Pumpe := "Panel".FP_CM01.Drucktest_Pumpe.Solldruck;
       "FP_CM01.GP01".Param.DT_Testzeit_Pumpe := DINT_TO_TIME(INT_TO_DINT("Panel".FP_CM01.Drucktest_Pumpe.Sollzeit) * 1000);
       // Drucktest Filter
       "FP_CM01.GP01".Param.DT_Druckaufbau := T#1m;
       "FP_CM01.GP01".Param.SW_Drucktest_Filter := "Panel".FP_CM01.Drucktest_Filter.Solldruck;
       "FP_CM01.GP01".Param.DT_Testzeit_Filter := DINT_TO_TIME(INT_TO_DINT("Panel".FP_CM01.Drucktest_Filter.Sollzeit) * 1000);

       IF "Panel".HQ01.Quitt_FW THEN
           "FP_CM01.GP01".In.Quitt_FW := TRUE;
           "Panel".HQ01.Quitt_FW := FALSE;
       END_IF;

       //--> Panel
       "Panel".CM01.GW_p_FP := "FP_CM01.GP01".Mld.GW_p_FP;
       "Panel".CM01.GW_LF_FP := "FP_CM01.GP01".Mld.GW_LF_FP;

       "Panel".FP_CM01.Sp_Ventil.Restzeit := TIME_TO_INT("FP_CM01.GP01".Zst.Restzeit_Spülen_Pumpe / 1000);
       "Panel".FP_CM01.Sp_Filter.Restzeit := TIME_TO_INT("FP_CM01.GP01".Zst.Restzeit_Filter / 1000);
       "Panel".FP_CM01.Drucktest_Pumpe.Restzeit := TIME_TO_INT("FP_CM01.GP01".Zst.Restzeit_DT / 1000);
       "Panel".FP_CM01.Drucktest_Pumpe.Schritt := "FP_CM01.GP01".Zst.Status_DT_Pumpe;
       "Panel".FP_CM01.Status_FW := "FP_CM01.GP01".Zst.Status_FW;

       "Panel".FP_CM01.Bedienung_Erlaubt := "FP_CM01.GP01".Zst.Bedienung_erlaubt;

       "Panel".FP_CM01.Status := "FP_CM01.GP01".Zst.Status_GP0x;
       "Panel".FP_CM01.speed := "FP_CM01.GP01".Zst.speed;

       "Panel".HQ01.S_Dkl_FG_li := "FP_CM01.GP01".In.Sensor_FG_links;
       "Panel".HQ01.S_Dkl_FG_re := "FP_CM01.GP01".In.Sensor_FG_rechts;
       "Panel".HQ01.S_FG_zu := "FP_CM01.GP01".In.Einhausung_HQ0x_zu;
       "Panel".HQ01.Niv_Leckage := NOT "FP_CM01.GP01".In.Leckage_ok;
       "Panel".HQ01.Quitt_FW_erlaubt := "FP_CM01.GP01".In.Sensor_FG_links AND "FP_CM01.GP01".In.Sensor_FG_rechts AND
       "FP_CM01.GP01".In.Einhausung_HQ0x_zu AND "FP_CM01.GP01".Mld.FG_Spülen_Ende AND "FP_CM01.GP01".Zst.Status_FW = 5;

       "Panel".FP_CM01.Drucktest_Filter.Restzeit := TIME_TO_INT("FP_CM01.GP01".Zst.Restzeit_DT / 1000);
       "Panel".FP_CM01.Drucktest_Filter.Schritt := "FP_CM01.GP01".Zst.Status_DT_Filter;
   END_REGION

   REGION Umwälzen
       "UP_CM01.GP02".Param.Name := 'UP_CM01.GP02';
       // Niveaus
       "UP_CM01.GP02".In.Niv_TLS := "E_Niv_TLS_CM01.BL04";
       "UP_CM01.GP02".In.Niv_min := "E_Niv_Min_CM01.BL03";
       "UP_CM01.GP02".In.Niv_max := "E_Niv_Max_CM01.BL02";
       "UP_CM01.GP02".In.Niv_Uel := NOT "E_Niv_UeL_CM01.BL01";
       "UP_CM01.GP02".In.Frg_Niv_CM05 := NOT "Pu_CM05.GP11_DB".In."Niv_max_CM05.BL01" AND NOT "Pu_CM05.GP11_DB".In."Niv_Uel_CM05.BL05";
       "UP_CM01.GP02".In.ext_Freigabe := "E_Al_Gas_ok" AND NOT "E_Not-Strom";
       // Ist-Druck
       "UP_CM01.GP02".In.Druck_Pumpe := "Panel".IW."p_CM01.BP04";

       //Stellrückmeldungen (Umwälzen)
       "UP_CM01.GP02".In.SRM_Saugseite_auf := "E_SRM_CM01.QM25_auf" AND NOT "E_SRM_CM01.QM25_zu";
       "UP_CM01.GP02".In.SRM_Saugseite_zu := "E_SRM_CM01.QM25_zu" AND NOT "E_SRM_CM01.QM25_auf";
       "UP_CM01.GP02".In.SRM_Druckseite_auf := "E_SRM_CM01.QM26_auf" AND NOT "E_SRM_CM01.QM26_zu";
       "UP_CM01.GP02".In.SRM_Druckseite_zu := "E_SRM_CM01.QM26_zu" AND NOT "E_SRM_CM01.QM26_auf";
       "UP_CM01.GP02".In.SRM_Eingang_Spülltg_auf := "E_SRM_CM01.QM20_auf" AND NOT "E_SRM_CM01.QM20_zu";
       "UP_CM01.GP02".In.SRM_Eingang_Spülltg_zu := "E_SRM_CM01.QM20_zu" AND NOT "E_SRM_CM01.QM20_auf";
       "UP_CM01.GP02".In.SRM_Ausgang_Spülltg_auf := "E_SRM_CM01.QM27_auf" AND NOT "E_SRM_CM01.QM27_zu";
       "UP_CM01.GP02".In.SRM_Ausgang_Spülltg_zu := "E_SRM_CM01.QM27_zu" AND NOT "E_SRM_CM01.QM27_auf";
       "UP_CM01.GP02".In.SRM_Entsogung_UV02_auf := "E_SRM_GP02.QM45_auf" AND NOT "E_SRM_GP02.QM45_zu";
       "UP_CM01.GP02".In.SRM_Entsogung_UV02_zu := "E_SRM_GP02.QM45_zu" AND NOT "E_SRM_GP02.QM45_auf";
       "UP_CM01.GP02".In.SRM_UV02_GP01_auf := "DB_PNOZ_IN_Out".In."SRM_Auf_BG-QM44" AND NOT "DB_PNOZ_IN_Out".In."SRM_Zu_BG-QM44";
       "UP_CM01.GP02".In.SRM_UV02_GP01_zu := "DB_PNOZ_IN_Out".In."SRM_Zu_BG-QM44" AND NOT "DB_PNOZ_IN_Out".In."SRM_Auf_BG-QM44";
       "UP_CM01.GP02".In.SRM_UV02_GP02_auf := "DB_PNOZ_IN_Out".In."SRM_Auf_BG-QM43" AND NOT "DB_PNOZ_IN_Out".In."SRM_Zu_BG-QM43";
       "UP_CM01.GP02".In.SRM_UV02_GP02_zu := "DB_PNOZ_IN_Out".In."SRM_Zu_BG-QM43" AND NOT "DB_PNOZ_IN_Out".In."SRM_Auf_BG-QM43";
       "UP_CM01.GP02".In."SRM_GP02.QM41_auf" := "E_SRM_GP02.QM41_auf" AND NOT "E_SRM_GP02.QM41_zu";
       "UP_CM01.GP02".In."SRM_GP01.QM14_auf" := "E_SRM_GP01.QM14_auf" AND NOT "E_SRM_GP01.QM14_zu";

       // Türen GP0x
       "UP_CM01.GP02".In.Tuer_zu_Seite_GP01 := "DB_PNOZ_IN_Out".In.Tuer_zu_Seite_GP01;
       "UP_CM01.GP02".In.Tuer_zu_vorn_GP01 := "DB_PNOZ_IN_Out".In.Tuer_zu_vorn_GP01;
       "UP_CM01.GP02".In.Tuer_zu_vorn_GP02 := "DB_PNOZ_IN_Out".In.Tuer_zu_vorn_GP02;
       // Leckagen Entsorgung
       "UP_CM01.GP02".In.Leckage_Doppelrohr_ok_BL26 := "E_LS_GP02.BL26";
       "UP_CM01.GP02".In.Leckage_Doppelschlauch_ok_BL33 := "E_LS_GP02.BL33";
       "UP_CM01.GP02".In.Leckage_Uml_Tunnel_ok_BL34 := "E_LS_GP01.BL34";
       "UP_CM01.GP02".In.Leckage_PFA_Uebergang_ok_BL16 := "E_LS_GP01.BL16";
       "UP_CM01.GP02".In.Leckage_PFA_Uebergang_ok_BL25 := "E_LS_GP02.BL25";

       "UP_CM01.GP02".In.Imp_Dfl := "E_Imp_GP02.BF02";
       "UP_CM01.GP02".In.Quitt_Al_Dfl := "DB_ANLAGE".IN.Quitt_Err;

       "UP_CM01.GP02".In.GW_p_UP := "E_GW_p_CM01.BP04";
       "UP_CM01.GP02".In.GW_LF_UP := "E_GW_LF_CM01.BN02";
       "UP_CM01.GP02".In.GW_Dfl := "E_GW_Dfl_GP02.BF02";
       // TW senkt
       "UP_CM01.GP02".In.TW_senkt := ("DB_POS".POS[1].FW_Senkt OR "DB_POS".POS[2].FW_Senkt OR "DB_POS".POS[3].FW_Senkt
       OR "DB_POS".POS[4].FW_Senkt OR "DB_POS".POS[5].FW_Senkt OR "DB_POS".POS[6].FW_Senkt) AND "DI_FW_1".ZST.Mittig;

       // Frequenzumrichter [Index 2] Umwälzen
       "UP_CM01.GP02".In.FU_speed := "FU_In_Out".FU[2].PE.Speed;
       "UP_CM01.GP02".In.FU_betriebsbereit := "FU_In_Out".FU[2].PE.Statusbyte.Bereit;
       "UP_CM01.GP02".In.FU_Stoerung := "FU_In_Out".FU[2].PE.Statusbyte.Stoer;
       "UP_CM01.GP02".Param.SW_Hand := "Panel".UP_CM01.SW_Hand;
       "UP_CM01.GP02".Param.SW_Auto_AZ := "Panel".UP_CM01.SW_Auto_AZ;
       "UP_CM01.GP02".Param.SW_Auto_aAZ := "Panel".UP_CM01.SW_Auto_aAZ;

       // Hand
       "UP_CM01.GP02".In.Ein := "Panel".UP_CM01.Ein;
       // Auto
       "UP_CM01.GP02".In.Auto := "Panel".UP_CM01.Auto;
       // Betriebsart
       "UP_CM01.GP02".In.Betriebsart := "Panel".UP_CM01.BA;
       // Spülzeit
       "UP_CM01.GP02".Param.Spülzeit := DINT_TO_TIME(INT_TO_DINT("Panel".UP_CM01.Sp_Ventil.Sollzeit) * 1000);
       // Drucktest
       "UP_CM01.GP02".Param.DT_Druckaufbau := T#1m;
       "UP_CM01.GP02".Param.SW_Drucktest := "Panel".UP_CM01.Drucktest.Solldruck;
       "UP_CM01.GP02".Param.DT_Testzeit := DINT_TO_TIME(INT_TO_DINT("Panel".UP_CM01.Drucktest.Sollzeit) * 1000);

       //--> Panel
       "Panel".CM01.Niv_TGS := "UP_CM01.GP02".In.Niv_TLS;
       "Panel".CM01.Niv_Min := "UP_CM01.GP02".In.Niv_min;
       "Panel".CM01.Niv_max := "UP_CM01.GP02".In.Niv_max;
       "Panel".CM01.Niv_Uel := "UP_CM01.GP02".Mld.Niv_Ueberlauf;
       "Panel".CM01.GW_p_UP := "UP_CM01.GP02".Mld.GW_p_UP;
       "Panel".CM01.GW_LF_UP := "UP_CM01.GP02".Mld.GW_LF_UP;
       "Panel".CM01.Niv_Proz := "UP_CM01.GP02".Zst.Niveau;
       "Panel".UP_CM01.Sp_Ventil.Restzeit := TIME_TO_INT("UP_CM01.GP02".Zst.Restzeit_Spülen / 1000);
       "Panel".UP_CM01.Drucktest.Restzeit := TIME_TO_INT("UP_CM01.GP02".Zst.Restzeit_DT / 1000);
       "Panel".UP_CM01.Drucktest.Schritt := "UP_CM01.GP02".Zst.Status_DT;
       "Panel".UP_CM01.Status := "UP_CM01.GP02".Zst.Status_GP0x;
       "Panel".UP_CM01.speed := "UP_CM01.GP02".Zst.speed;
       "Panel".UP_CM01.Bedienung_Erlaubt := "UP_CM01.GP02".Zst.Bedienung_erlaubt;
   END_REGION
END_REGION

REGION Network 4 (SCL): CM02
   REGION Filtern
       "FP_CM02.GP04".Param.Name_Pumpe := 'FP_CM02.GP04';
       "FP_CM02.GP04".Param.Name_Filter := 'Filter HQ2';
       // Niveaus
       "FP_CM02.GP04".In.Niv_TLS := "E_Niv_TLS_CM02.BL11";
       "FP_CM02.GP04".In.Niv_min := "E_Niv_Min_CM02.BL10";
       "FP_CM02.GP04".In.Niv_max := "E_Niv_Max_CM02.BL09";
       "FP_CM02.GP04".In.Niv_Uel := NOT "E_Niv_UeL_CM02.BL08";
       "FP_CM02.GP04".In.Frg_Niv_CM05 := NOT "Pu_CM05.GP11_DB".In."Niv_max_CM05.BL01" AND NOT "Pu_CM05.GP11_DB".In."Niv_Uel_CM05.BL05";
       "FP_CM02.GP04".In.Leckage_ok := "E_LS_HQ0x.BL12";
       "FP_CM02.GP04".In.ext_Freigabe := "E_Al_Gas_ok" AND NOT "E_Not-Strom";
       // Ist-Druck Pumpe
       "FP_CM02.GP04".In.Druck_Pumpe := "Panel".IW."p_CM02.BP06";
       // Differenz-Druck Filter
       "FP_CM02.GP04".In.Delta_p_Filter := "Panel".IW."p_HQ02.BP02";

       //Stellrückmeldungen (Filtern)
       "FP_CM02.GP04".In.SRM_Saugseite_auf := "E_SRM_CM02.QM55_auf" AND NOT "E_SRM_CM02.QM55_zu";
       "FP_CM02.GP04".In.SRM_Saugseite_zu := "E_SRM_CM02.QM55_zu" AND NOT "E_SRM_CM02.QM55_auf";
       "FP_CM02.GP04".In.SRM_Eingang_Filter_auf := "E_SRM_HQ02.QM59_auf" AND NOT "E_SRM_HQ02.QM59_zu";
       "FP_CM02.GP04".In.SRM_Eingang_Filter_zu := "E_SRM_HQ02.QM59_zu" AND NOT "E_SRM_HQ02.QM59_auf";
       "FP_CM02.GP04".In.SRM_Ausgang_Filter_auf := "E_SRM_HQ02.QM60_auf" AND NOT "E_SRM_HQ02.QM60_zu";
       "FP_CM02.GP04".In.SRM_Ausgang_Filter_zu := "E_SRM_HQ02.QM60_zu" AND NOT "E_SRM_HQ02.QM60_auf";

       "FP_CM02.GP04".In.SRM_Eingang_Spülltg_P_auf := "E_SRM_CM02.QM56_auf" AND NOT "E_SRM_CM02.QM56_zu";
       "FP_CM02.GP04".In.SRM_Eingang_Spülltg_P_zu := "E_SRM_CM02.QM56_zu" AND NOT "E_SRM_CM02.QM56_auf";
       "FP_CM02.GP04".In.SRM_Eingang_Spülltg_F_auf := "E_SRM_HQ02.QM58_auf" AND NOT "E_SRM_HQ02.QM58_zu";
       "FP_CM02.GP04".In.SRM_Eingang_Spülltg_F_zu := "E_SRM_HQ02.QM58_zu" AND NOT "E_SRM_HQ02.QM58_auf";
       "FP_CM02.GP04".In.SRM_Ausgang_Spülltg_auf := "E_SRM_HQ02.QM61_auf" AND NOT "E_SRM_HQ02.QM61_zu";
       "FP_CM02.GP04".In.SRM_Ausgang_Spülltg_zu := "E_SRM_HQ02.QM61_zu" AND NOT "E_SRM_HQ02.QM61_auf";
       "FP_CM02.GP04".In.SRM_Entluften_auf := "E_SRM_HQ02.LV02_auf" AND NOT "E_SRM_HQ02.LV02_zu";
       "FP_CM02.GP04".In.SRM_Entlueften_zu := "E_SRM_HQ02.LV02_zu" AND NOT "E_SRM_HQ02.LV02_auf";

       // Filtergehäuse
       "FP_CM02.GP04".In.GW_p_FG := "E_GW_p_HQ02.BP02";
       "FP_CM02.GP04".In.Sensor_FG_links := "E_S_FG_li_HQ02.BG10";
       "FP_CM02.GP04".In.Sensor_FG_rechts := "E_S_FG_re_HQ02.BG11";
       "FP_CM02.GP04".In.Einhausung_HQ0x_zu := "DB_PNOZ_IN_Out".In.FG_zu_HQ02;
       "FP_CM02.GP04".Param.WarnGr_FW := "Panel".HQ02.WarnGr_FW;
       "FP_CM02.GP04".Param.Wechsel_FW := "Panel".HQ02.Wechsel_FW;

       // Not-Halt
       "FP_CM02.GP04".In.NotHalt := NOT "DB_PNOZ_IN_Out".In.NH_Frg_FP_CM02;

       "FP_CM02.GP04".In.GW_p_FP := "E_GW_p_CM02.BP06";
       "FP_CM02.GP04".In.GW_LF_FP := "E_GW_LF_CM02.BN03";

       // Frequenzumrichter [Index 4] 
       "FP_CM02.GP04".In.FU_speed := "FU_In_Out".FU[4].PE.Speed;
       "FP_CM02.GP04".In.FU_betriebsbereit := "FU_In_Out".FU[4].PE.Statusbyte.Bereit;
       "FP_CM02.GP04".In.FU_Stoerung := "FU_In_Out".FU[4].PE.Statusbyte.Stoer;
       "FP_CM02.GP04".Param.SW_Hand := "Panel".FP_CM02.SW_Hand;
       "FP_CM02.GP04".Param.SW_Auto_AZ := "Panel".FP_CM02.SW_Auto_AZ;
       "FP_CM02.GP04".Param.SW_Auto_aAZ := "Panel".FP_CM02.SW_Auto_aAZ;

       // Hand
       "FP_CM02.GP04".In.Ein := "Panel".FP_CM02.Ein;
       // Auto
       "FP_CM02.GP04".In.Auto := "Panel".FP_CM02.Auto;
       // Betriebsart
       "FP_CM02.GP04".In.Betriebsart := "Panel".FP_CM02.BA;
       // Spülzeit
       "FP_CM02.GP04".Param.Spülzeit_Pumpe := DINT_TO_TIME(INT_TO_DINT("Panel".FP_CM02.Sp_Ventil.Sollzeit) * 1000);
       // Zeiten Filterwechsel
       "FP_CM02.GP04".Param.FG_Zeit_leeren_Saurebecken := DINT_TO_TIME(INT_TO_DINT("Panel".FP_CM02.Sp_Filter.Zeit_leeren_Saure) * 1000);
       "FP_CM02.GP04".Param.FG_Zeit_leeren_CM05 := DINT_TO_TIME(INT_TO_DINT("Panel".FP_CM02.Sp_Filter.Zeit_leeren_CM05) * 1000);
       "FP_CM02.GP04".Param.FW_Spülzeit := DINT_TO_TIME(INT_TO_DINT("Panel".FP_CM02.Sp_Filter.Zeit_Spülen) * 1000);
       "FP_CM02.GP04".Param.FW_Wartezeit := DINT_TO_TIME(INT_TO_DINT("Panel".FP_CM02.Sp_Filter.Wartezeit) * 1000);
       "FP_CM02.GP04".Param.FW_Zeit_fuellen := DINT_TO_TIME(INT_TO_DINT("Panel".FP_CM02.Sp_Filter.Zeit_füllen) * 1000);
       "Panel".FP_CM02.Status_FW := "FP_CM02.GP04".Zst.Status_FW;
       // Drucktest Pumpe
       "FP_CM02.GP04".Param.DT_Druckaufbau := T#1m;
       "FP_CM02.GP04".Param.SW_Drucktest_Pumpe := "Panel".FP_CM02.Drucktest_Pumpe.Solldruck;
       "FP_CM02.GP04".Param.DT_Testzeit_Pumpe := DINT_TO_TIME(INT_TO_DINT("Panel".FP_CM02.Drucktest_Pumpe.Sollzeit) * 1000);
       // Drucktest Filter
       "FP_CM02.GP04".Param.DT_Druckaufbau := T#1m;
       "FP_CM02.GP04".Param.SW_Drucktest_Filter := "Panel".FP_CM02.Drucktest_Filter.Solldruck;
       "FP_CM02.GP04".Param.DT_Testzeit_Filter := DINT_TO_TIME(INT_TO_DINT("Panel".FP_CM02.Drucktest_Filter.Sollzeit) * 1000);

       IF "Panel".HQ02.Quitt_FW THEN
           "FP_CM02.GP04".In.Quitt_FW := TRUE;
           "Panel".HQ02.Quitt_FW := FALSE;
       END_IF;

       //--> Panel
       "Panel".CM02.GW_p_FP := "FP_CM02.GP04".Mld.GW_p_FP;
       "Panel".CM02.GW_LF_FP := "FP_CM02.GP04".Mld.GW_LF_FP;

       "Panel".FP_CM02.Sp_Ventil.Restzeit := TIME_TO_INT("FP_CM02.GP04".Zst.Restzeit_Spülen_Pumpe / 1000);
       "Panel".FP_CM02.Sp_Filter.Restzeit := TIME_TO_INT("FP_CM02.GP04".Zst.Restzeit_Filter / 1000);
       "Panel".FP_CM02.Drucktest_Pumpe.Restzeit := TIME_TO_INT("FP_CM02.GP04".Zst.Restzeit_DT / 1000);
       "Panel".FP_CM02.Drucktest_Pumpe.Schritt := "FP_CM02.GP04".Zst.Status_DT_Pumpe;
       "Panel".FP_CM02.Status := "FP_CM02.GP04".Zst.Status_GP0x;
       "Panel".FP_CM02.speed := "FP_CM02.GP04".Zst.speed;

       "Panel".FP_CM02.Bedienung_Erlaubt := "FP_CM02.GP04".Zst.Bedienung_erlaubt;

       "Panel".HQ02.S_Dkl_FG_li := "FP_CM02.GP04".In.Sensor_FG_links;
       "Panel".HQ02.S_Dkl_FG_re := "FP_CM02.GP04".In.Sensor_FG_rechts;
       "Panel".HQ02.S_FG_zu := "FP_CM02.GP04".In.Einhausung_HQ0x_zu;
       "Panel".HQ02.Niv_Leckage := NOT "FP_CM02.GP04".In.Leckage_ok;

       "Panel".HQ02.Quitt_FW_erlaubt := "FP_CM02.GP04".In.Sensor_FG_links AND "FP_CM02.GP04".In.Sensor_FG_rechts AND
       "FP_CM02.GP04".In.Einhausung_HQ0x_zu AND "FP_CM02.GP04".Mld.FG_Spülen_Ende AND "FP_CM02.GP04".Zst.Status_FW = 5;

       "Panel".FP_CM02.Drucktest_Filter.Restzeit := TIME_TO_INT("FP_CM02.GP04".Zst.Restzeit_DT / 1000);
       "Panel".FP_CM02.Drucktest_Filter.Schritt := "FP_CM02.GP04".Zst.Status_DT_Filter;
   END_REGION

   REGION Umwälzen
       "UP_CM02.GP05".Param.Name := 'UP_CM02.GP05';
       // Niveaus
       "UP_CM02.GP05".In.Niv_TLS := "E_Niv_TLS_CM02.BL11";
       "UP_CM02.GP05".In.Niv_min := "E_Niv_Min_CM02.BL10";
       "UP_CM02.GP05".In.Niv_max := "E_Niv_Max_CM02.BL09";
       "UP_CM02.GP05".In.Niv_Uel := NOT "E_Niv_UeL_CM02.BL08";
       "UP_CM02.GP05".In.Frg_Niv_CM05 := NOT "Pu_CM05.GP11_DB".In."Niv_max_CM05.BL01" AND NOT "Pu_CM05.GP11_DB".In."Niv_Uel_CM05.BL05";
       "UP_CM02.GP05".In.ext_Freigabe := "E_Al_Gas_ok" AND NOT "E_Not-Strom";
       // Ist-Druck
       "UP_CM02.GP05".In.Druck_Pumpe := "Panel".IW."p_CM02.BP07";

       //Stellrückmeldungen
       "UP_CM02.GP05".In.SRM_Saugseite_auf := "E_SRM_CM02.QM62_auf" AND NOT "E_SRM_CM02.QM62_zu";
       "UP_CM02.GP05".In.SRM_Saugseite_zu := "E_SRM_CM02.QM62_zu" AND NOT "E_SRM_CM02.QM62_auf";
       "UP_CM02.GP05".In.SRM_Druckseite_auf := "E_SRM_CM02.QM63_auf" AND NOT "E_SRM_CM02.QM63_zu";
       "UP_CM02.GP05".In.SRM_Druckseite_zu := "E_SRM_CM02.QM63_zu" AND NOT "E_SRM_CM02.QM63_auf";
       "UP_CM02.GP05".In.SRM_Eingang_Spülltg_auf := "E_SRM_CM02.QM57_auf" AND NOT "E_SRM_CM02.QM57_zu";
       "UP_CM02.GP05".In.SRM_Eingang_Spülltg_zu := "E_SRM_CM02.QM57_zu" AND NOT "E_SRM_CM02.QM57_auf";
       "UP_CM02.GP05".In.SRM_Ausgang_Spülltg_auf := "E_SRM_CM02.QM64_auf" AND NOT "E_SRM_CM02.QM64_zu";
       "UP_CM02.GP05".In.SRM_Ausgang_Spülltg_zu := "E_SRM_CM02.QM64_zu" AND NOT "E_SRM_CM02.QM64_auf";
       "UP_CM02.GP05".In.SRM_Entsogung_UV02_auf := "E_SRM_GP02.QM46_auf" AND NOT "E_SRM_GP02.QM46_zu";
       "UP_CM02.GP05".In.SRM_Entsogung_UV02_zu := "E_SRM_GP02.QM46_zu" AND NOT "E_SRM_GP02.QM46_auf";
       "UP_CM02.GP05".In.SRM_UV02_GP01_auf := "DB_PNOZ_IN_Out".In."SRM_Auf_BG-QM44" AND NOT "DB_PNOZ_IN_Out".In."SRM_Zu_BG-QM44";
       "UP_CM02.GP05".In.SRM_UV02_GP01_zu := "DB_PNOZ_IN_Out".In."SRM_Zu_BG-QM44" AND NOT "DB_PNOZ_IN_Out".In."SRM_Auf_BG-QM44";
       "UP_CM02.GP05".In.SRM_UV02_GP02_auf := "DB_PNOZ_IN_Out".In."SRM_Auf_BG-QM43" AND NOT "DB_PNOZ_IN_Out".In."SRM_Zu_BG-QM43";
       "UP_CM02.GP05".In.SRM_UV02_GP02_zu := "DB_PNOZ_IN_Out".In."SRM_Zu_BG-QM43" AND NOT "DB_PNOZ_IN_Out".In."SRM_Auf_BG-QM43";
       "UP_CM02.GP05".In."SRM_GP02.QM41_auf" := "E_SRM_GP02.QM41_auf" AND NOT "E_SRM_GP02.QM41_zu";
       "UP_CM02.GP05".In."SRM_GP01.QM14_auf" := "E_SRM_GP01.QM14_auf" AND NOT "E_SRM_GP01.QM14_zu";

       // Türen GP0x
       "UP_CM02.GP05".In.Tuer_zu_Seite_GP01 := "DB_PNOZ_IN_Out".In.Tuer_zu_Seite_GP01;
       "UP_CM02.GP05".In.Tuer_zu_vorn_GP01 := "DB_PNOZ_IN_Out".In.Tuer_zu_vorn_GP01;
       "UP_CM02.GP05".In.Tuer_zu_vorn_GP02 := "DB_PNOZ_IN_Out".In.Tuer_zu_vorn_GP02;

       // Leckagen Entsorgung
       "UP_CM02.GP05".In.Leckage_Doppelrohr_ok_BL26 := "E_LS_GP02.BL26";
       "UP_CM02.GP05".In.Leckage_Doppelschlauch_ok_BL33 := "E_LS_GP02.BL33";
       "UP_CM02.GP05".In.Leckage_Uml_Tunnel_ok_BL34 := "E_LS_GP01.BL34";
       "UP_CM02.GP05".In.Leckage_PFA_Uebergang_ok_BL16 := "E_LS_GP01.BL16";
       "UP_CM02.GP05".In.Leckage_PFA_Uebergang_ok_BL25 := "E_LS_GP02.BL25";

       "UP_CM02.GP05".In.Imp_Dfl := "E_Imp_GP02.BF02";
       "UP_CM02.GP05".In.Quitt_Al_Dfl := "DB_ANLAGE".IN.Quitt_Err;

       "UP_CM02.GP05".In.GW_p_UP := "E_GW_p_CM02.BP07";
       "UP_CM02.GP05".In.GW_p_UP := "E_GW_LF_CM02.BN04";
       "UP_CM02.GP05".In.GW_Dfl := "E_GW_Dfl_GP02.BF02";
       // TW senkt
       "UP_CM02.GP05".In.TW_senkt := ("DB_POS".POS[13].FW_Senkt OR "DB_POS".POS[14].FW_Senkt OR "DB_POS".POS[15].FW_Senkt
       OR "DB_POS".POS[16].FW_Senkt OR "DB_POS".POS[17].FW_Senkt OR "DB_POS".POS[18].FW_Senkt) AND "DI_FW_1".ZST.Mittig;

       // Frequenzumrichter [Index 5]
       "UP_CM02.GP05".In.FU_speed := "FU_In_Out".FU[5].PE.Speed;
       "UP_CM02.GP05".In.FU_betriebsbereit := "FU_In_Out".FU[5].PE.Statusbyte.Bereit;
       "UP_CM02.GP05".In.FU_Stoerung := "FU_In_Out".FU[5].PE.Statusbyte.Stoer;
       "UP_CM02.GP05".Param.SW_Hand := "Panel".UP_CM02.SW_Hand;
       "UP_CM02.GP05".Param.SW_Auto_AZ := "Panel".UP_CM02.SW_Auto_AZ;
       "UP_CM02.GP05".Param.SW_Auto_aAZ := "Panel".UP_CM02.SW_Auto_aAZ;

       // Hand
       "UP_CM02.GP05".In.Ein := "Panel".UP_CM02.Ein;
       // Auto
       "UP_CM02.GP05".In.Auto := "Panel".UP_CM02.Auto;
       // Betriebsart
       "UP_CM02.GP05".In.Betriebsart := "Panel".UP_CM02.BA;
       // Spülzeit
       "UP_CM02.GP05".Param.Spülzeit := DINT_TO_TIME(INT_TO_DINT("Panel".UP_CM02.Sp_Ventil.Sollzeit) * 1000);
       // Drucktest
       "UP_CM02.GP05".Param.DT_Druckaufbau := T#1m;
       "UP_CM02.GP05".Param.SW_Drucktest := "Panel".UP_CM02.Drucktest.Solldruck;
       "UP_CM02.GP05".Param.DT_Testzeit := DINT_TO_TIME(INT_TO_DINT("Panel".UP_CM02.Drucktest.Sollzeit) * 1000);

       //--> Panel
       "Panel".CM02.Niv_TGS := "UP_CM02.GP05".In.Niv_TLS;
       "Panel".CM02.Niv_Min := "UP_CM02.GP05".In.Niv_min;
       "Panel".CM02.Niv_max := "UP_CM02.GP05".In.Niv_max;
       "Panel".CM02.Niv_Uel := "UP_CM02.GP05".Mld.Niv_Ueberlauf;
       "Panel".CM02.GW_p_UP := "UP_CM02.GP05".Mld.GW_p_UP;
       "Panel".CM02.GW_LF_UP := "UP_CM02.GP05".Mld.GW_LF_UP;
       "Panel".CM02.Niv_Proz := "UP_CM02.GP05".Zst.Niveau;
       "Panel".UP_CM02.Sp_Ventil.Restzeit := TIME_TO_INT("UP_CM02.GP05".Zst.Restzeit_Spülen / 1000);
       "Panel".UP_CM02.Drucktest.Restzeit := TIME_TO_INT("UP_CM02.GP05".Zst.Restzeit_DT / 1000);
       "Panel".UP_CM02.Drucktest.Schritt := "UP_CM02.GP05".Zst.Status_DT;
       "Panel".UP_CM02.Status := "UP_CM02.GP05".Zst.Status_GP0x;
       "Panel".UP_CM02.speed := "UP_CM02.GP05".Zst.speed;
       "Panel".UP_CM02.Bedienung_Erlaubt := "UP_CM02.GP05".Zst.Bedienung_erlaubt;
   END_REGION
END_REGION

REGION Network 5 (SCL): CM03
   "UP_CM03.GP03".Param.Name := 'UP_CM03.GP03';
   // Niveaus
   "UP_CM03.GP03".In.Niv_TLS := "E_Niv_TLS_CM03.BL07";
   "UP_CM03.GP03".In.Niv_min := "E_Niv_Min_CM03.BL06";
   "UP_CM03.GP03".In.Frg_Niv_CM05 := NOT "Pu_CM05.GP11_DB".In."Niv_max_CM05.BL01" AND NOT "Pu_CM05.GP11_DB".In."Niv_Uel_CM05.BL05";
   "UP_CM03.GP03".In.ext_Freigabe := "E_Al_Gas_ok" AND NOT"E_Not-Strom";
   // Ist-Druck
   "UP_CM03.GP03".In.Druck_Pumpe := "Panel".IW."p_CM03.BP05";

